LIN {X 0,Y 453.948,Z 433.148,A -85,B 0,C 180,E1 19620.953,E2 19620.953} C_VEL
LIN {X 0,Y 449.947,Z 427.727,A -85,B 0,C 180,E1 19618.536,E2 19618.536} C_VEL
LIN {X 0,Y 445.616,Z 421.973,A -85,B 0,C 180,E1 19615.625,E2 19615.625} C_VEL
LIN {X 0,Y 442.629,Z 417.979,A -85,B 0,C 180,E1 19613.319,E2 19613.319} C_VEL
LIN {X 0,Y 441.414,Z 416.212,A -85,B 0,C 180,E1 19612.32,E2 19612.32} C_VEL
LIN {X 0,Y 438.487,Z 412.431,A -85,B 0,C 180,E1 19609.754,E2 19609.754} C_VEL
LIN {X 0,Y 437.49,Z 410.574,A -85,B 0,C 180,E1 19608.658,E2 19608.658} C_VEL
LIN {X 0,Y 434.499,Z 406.882,A -85,B 0,C 180,E1 19605.473,E2 19605.473} C_VEL
LIN {X 0,Y 433.389,Z 405.057,A -85,B 0,C 180,E1 19604.065,E2 19604.065} C_VEL
LIN {X 0,Y 430.291,Z 402.854,A -85,B 0,C 180,E1 19600.026,E2 19600.026} C_VEL
LIN {X 0,Y 428.498,Z 399.899,A -85,B 0,C 180,E1 19596.497,E2 19596.497} C_VEL
LIN {X 0,Y 427.919,Z 398.821,A -85,B 0,C 180,E1 19594.98,E2 19594.98} C_VEL
LIN {X 0,Y 426.399,Z 397.892,A -85,B 0,C 180,E1 19590.961,E2 19590.961} C_VEL
LIN {X 0,Y 425.533,Z 397.406,A -85,B 0,C 180,E1 19586.482,E2 19586.482} C_VEL
LIN {X 0,Y 425.524,Z 397.366,A -85,B 0,C 180,E1 19581.704,E2 19581.704} C_VEL
LIN {X 0,Y 426.383,Z 397.854,A -85,B 0,C 180,E1 19577.222,E2 19577.222} C_VEL
LIN {X 0,Y 428.081,Z 398.875,A -85,B 0,C 180,E1 19573.002,E2 19573.002} C_VEL
LIN {X 0,Y 430.356,Z 402.874,A -85,B 0,C 180,E1 19568.465,E2 19568.465} C_VEL
LIN {X 0,Y 433.58,Z 405.087,A -85,B 0,C 180,E1 19564.562,E2 19564.562} C_VEL
LIN {X 0,Y 434.467,Z 405.993,A -85,B 0,C 180,E1 19563.639,E2 19563.639} C_VEL
LIN {X 0,Y 436.45,Z 409.448,A -85,B 0,C 180,E1 19561.412,E2 19561.412} C_VEL
LIN {X 0,Y 440.205,Z 412.266,A -85,B 0,C 180,E1 19558.341,E2 19558.341} C_VEL
LIN {X 0,Y 442.471,Z 415.992,A -85,B 0,C 180,E1 19556.507,E2 19556.507} C_VEL
LIN {X 0,Y 445.89,Z 418.808,A -85,B 0,C 180,E1 19554.263,E2 19554.263} C_VEL
LIN {X 0,Y 448.38,Z 422.573,A -85,B 0,C 180,E1 19552.597,E2 19552.597} C_VEL
LIN {X 0,Y 451.551,Z 425.296,A -85,B 0,C 180,E1 19550.859,E2 19550.859} C_VEL
LIN {X 0,Y 454.634,Z 429.505,A -85,B 0,C 180,E1 19549.129,E2 19549.129} C_VEL
LIN {X 0,Y 456.956,Z 431.699,A -85,B 0,C 180,E1 19548.003,E2 19548.003} C_VEL
LIN {X 0,Y 460.475,Z 436.08,A -85,B 0,C 180,E1 19546.306,E2 19546.306} C_VEL
LIN {X 0,Y 462.233,Z 437.873,A -85,B 0,C 180,E1 19545.527,E2 19545.527} C_VEL
LIN {X 0,Y 466.393,Z 442.761,A -85,B 0,C 180,E1 19543.767,E2 19543.767} C_VEL
LIN {X 0,Y 472.76,Z 450.553,A -85,B 0,C 180,E1 19541.251,E2 19541.251} C_VEL
LIN {X 0,Y 477.709,Z 456.627,A -85,B 0,C 180,E1 19539.457,E2 19539.457} C_VEL
LIN {X 0,Y 482.621,Z 462.669,A -85,B 0,C 180,E1 19537.805,E2 19537.805} C_VEL
LIN {X 0,Y 489.868,Z 471.652,A -85,B 0,C 180,E1 19535.534,E2 19535.534} C_VEL
LIN {X 0,Y 501.803,Z 487.082,A -85,B 0,C 180,E1 19532.17,E2 19532.17} C_VEL
LIN {X 0,Y 513.739,Z 503.433,A -85,B 0,C 180,E1 19529.164,E2 19529.164} C_VEL
LIN {X 0,Y 519.251,Z 511.432,A -85,B 0,C 180,E1 19527.864,E2 19527.864} C_VEL
LIN {X 0,Y 504.477,Z 710.205,A -85,B 0,C 180,E1 19524.562,E2 19524.562} C_VEL
LIN {X 0,Y 499.182,Z 782.061,A -85,B 0,C 180,E1 19523.337,E2 19523.337} C_VEL
LIN {X 0,Y 496,Z 810.118,A -85,B 0,C 180,E1 19522.672,E2 19522.672} C_VEL
LIN {X 0,Y 492.733,Z 832.872,A -85,B 0,C 180,E1 19521.983,E2 19521.983} C_VEL
LIN {X 0,Y 488.951,Z 855.104,A -85,B 0,C 180,E1 19521.169,E2 19521.169} C_VEL
LIN {X 0,Y 483.544,Z 882.162,A -85,B 0,C 180,E1 19519.967,E2 19519.967} C_VEL
LIN {X 0,Y 482.445,Z 886.921,A -85,B 0,C 180,E1 19519.725,E2 19519.725} C_VEL
LIN {X 0,Y 480.2,Z 894.101,A -85,B 0,C 180,E1 19519.451,E2 19519.451} C_VEL
LIN {X 0,Y 471.991,Z 912.002,A -85,B 0,C 180,E1 19519.007,E2 19519.007} C_VEL
LIN {X 0,Y 469.526,Z 918.813,A -85,B 0,C 180,E1 19518.673,E2 19518.673} C_VEL
LIN {X 0,Y 463.65,Z 939.58,A -85,B 0,C 180,E1 19517.251,E2 19517.251} C_VEL
LIN {X 0,Y 457.958,Z 958.139,A -85,B 0,C 180,E1 19515.794,E2 19515.794} C_VEL
LIN {X 0,Y 451.926,Z 976.561,A -85,B 0,C 180,E1 19514.149,E2 19514.149} C_VEL
LIN {X 0,Y 444.682,Z 997.402,A -85,B 0,C 180,E1 19512.016,E2 19512.016} C_VEL
LIN {X 0,Y 437.637,Z 1016.215,A -85,B 0,C 180,E1 19509.756,E2 19509.756} C_VEL
LIN {X 0,Y 431.782,Z 1031.379,A -85,B 0,C 180,E1 19507.68,E2 19507.68} C_VEL
LIN {X 0,Y 426.261,Z 1045.276,A -85,B 0,C 180,E1 19505.525,E2 19505.525} C_VEL
LIN {X 0,Y 420.181,Z 1060.321,A -85,B 0,C 180,E1 19502.873,E2 19502.873} C_VEL
LIN {X 0,Y 413.774,Z 1076.012,A -85,B 0,C 180,E1 19499.621,E2 19499.621} C_VEL
LIN {X 0,Y 409.258,Z 1087.2,A -85,B 0,C 180,E1 19496.931,E2 19496.931} C_VEL
LIN {X 0,Y 405.334,Z 1097.229,A -85,B 0,C 180,E1 19494.173,E2 19494.173} C_VEL
LIN {X 0,Y 401.802,Z 1106.699,A -85,B 0,C 180,E1 19491.161,E2 19491.161} C_VEL
LIN {X 0,Y 398.332,Z 1116.847,A -85,B 0,C 180,E1 19487.333,E2 19487.333} C_VEL
LIN {X 0,Y 396.087,Z 1124.106,A -85,B 0,C 180,E1 19483.965,E2 19483.965} C_VEL
LIN {X 0,Y 394.719,Z 1129.457,A -85,B 0,C 180,E1 19480.986,E2 19480.986} C_VEL
LIN {X 0,Y 393.77,Z 1133.759,A -85,B 0,C 180,E1 19478.079,E2 19478.079} C_VEL
LIN {X 0,Y 393.212,Z 1137.313,A -85,B 0,C 180,E1 19475.036,E2 19475.036} C_VEL
LIN {X 0,Y 392.895,Z 1140.115,A -85,B 0,C 180,E1 19471.789,E2 19471.789} C_VEL
LIN {X 0,Y 392.777,Z 1141.998,A -85,B 0,C 180,E1 19468.428,E2 19468.428} C_VEL
LIN {X 0,Y 392.756,Z 1142.857,A -85,B 0,C 180,E1 19464.518,E2 19464.518} C_VEL
LIN {X 0,Y 392.867,Z 1142.444,A -85,B 0,C 180,E1 19461.187,E2 19461.187} C_VEL
LIN {X 0,Y 393.077,Z 1141.179,A -85,B 0,C 180,E1 19458.08,E2 19458.08} C_VEL
LIN {X 0,Y 393.472,Z 1139.082,A -85,B 0,C 180,E1 19455.023,E2 19455.023} C_VEL
LIN {X 0,Y 394.158,Z 1136.173,A -85,B 0,C 180,E1 19452.006,E2 19452.006} C_VEL
LIN {X 0,Y 395.37,Z 1132.022,A -85,B 0,C 180,E1 19448.728,E2 19448.728} C_VEL
LIN {X 0,Y 397.737,Z 1125.255,A -85,B 0,C 180,E1 19444.614,E2 19444.614} C_VEL
LIN {X 0,Y 400.473,Z 1118.328,A -85,B 0,C 180,E1 19441.288,E2 19441.288} C_VEL
LIN {X 0,Y 403.679,Z 1110.94,A -85,B 0,C 180,E1 19438.297,E2 19438.297} C_VEL
LIN {X 0,Y 408.437,Z 1100.796,A -85,B 0,C 180,E1 19434.803,E2 19434.803} C_VEL
LIN {X 0,Y 414.124,Z 1088.742,A -85,B 0,C 180,E1 19431.391,E2 19431.391} C_VEL
LIN {X 0,Y 419.404,Z 1077.818,A -85,B 0,C 180,E1 19428.726,E2 19428.726} C_VEL
LIN {X 0,Y 426.356,Z 1063.666,A -85,B 0,C 180,E1 19425.744,E2 19425.744} C_VEL
LIN {X 0,Y 433.69,Z 1048.049,A -85,B 0,C 180,E1 19422.974,E2 19422.974} C_VEL
LIN {X 0,Y 440.644,Z 1033.015,A -85,B 0,C 180,E1 19420.652,E2 19420.652} C_VEL
LIN {X 0,Y 448.963,Z 1014.263,A -85,B 0,C 180,E1 19418.165,E2 19418.165} C_VEL
LIN {X 0,Y 456.181,Z 997.272,A -85,B 0,C 180,E1 19416.215,E2 19416.215} C_VEL
LIN {X 0,Y 464.592,Z 976.767,A -85,B 0,C 180,E1 19414.162,E2 19414.162} C_VEL
LIN {X 0,Y 473.151,Z 955.052,A -85,B 0,C 180,E1 19412.295,E2 19412.295} C_VEL
LIN {X 0,Y 483.358,Z 928.968,A -85,B 0,C 180,E1 19410.369,E2 19410.369} C_VEL
LIN {X 0,Y 492.594,Z 906.196,A -85,B 0,C 180,E1 19408.935,E2 19408.935} C_VEL
LIN {X 0,Y 480.962,Z 937.636,A -85,B 0,C 180,E1 19407.68,E2 19407.68} C_VEL
LIN {X 0,Y 469.639,Z 971.581,A -85,B 0,C 180,E1 19406.022,E2 19406.022} C_VEL
LIN {X 0,Y 459.445,Z 1005.778,A -85,B 0,C 180,E1 19404.054,E2 19404.054} C_VEL
LIN {X 0,Y 451.325,Z 1034.155,A -85,B 0,C 180,E1 19402.144,E2 19402.144} C_VEL
LIN {X 0,Y 444.279,Z 1059.225,A -85,B 0,C 180,E1 19400.225,E2 19400.225} C_VEL
LIN {X 0,Y 436.325,Z 1087.372,A -85,B 0,C 180,E1 19397.747,E2 19397.747} C_VEL
LIN {X 0,Y 430.123,Z 1109.071,A -85,B 0,C 180,E1 19395.533,E2 19395.533} C_VEL
LIN {X 0,Y 425.026,Z 1126.85,A -85,B 0,C 180,E1 19393.497,E2 19393.497} C_VEL
LIN {X 0,Y 420.318,Z 1143.268,A -85,B 0,C 180,E1 19391.401,E2 19391.401} C_VEL
LIN {X 0,Y 415.947,Z 1158.657,A -85,B 0,C 180,E1 19389.214,E2 19389.214} C_VEL
LIN {X 0,Y 411.781,Z 1173.547,A -85,B 0,C 180,E1 19386.853,E2 19386.853} C_VEL
LIN {X 0,Y 407.666,Z 1188.654,A -85,B 0,C 180,E1 19384.171,E2 19384.171} C_VEL
LIN {X 0,Y 403.227,Z 1205.646,A -85,B 0,C 180,E1 19380.718,E2 19380.718} C_VEL
LIN {X 0,Y 399.899,Z 1219.42,A -85,B 0,C 180,E1 19377.423,E2 19377.423} C_VEL
LIN {X 0,Y 397.604,Z 1230.079,A -85,B 0,C 180,E1 19374.515,E2 19374.515} C_VEL
LIN {X 0,Y 395.951,Z 1238.807,A -85,B 0,C 180,E1 19371.79,E2 19371.79} C_VEL
LIN {X 0,Y 394.633,Z 1246.816,A -85,B 0,C 180,E1 19368.924,E2 19368.924} C_VEL
LIN {X 0,Y 393.741,Z 1253.611,A -85,B 0,C 180,E1 19366.069,E2 19366.069} C_VEL
LIN {X 0,Y 393.177,Z 1259.28,A -85,B 0,C 180,E1 19363.231,E2 19363.231} C_VEL
LIN {X 0,Y 392.885,Z 1263.863,A -85,B 0,C 180,E1 19360.41,E2 19360.41} C_VEL
LIN {X 0,Y 392.748,Z 1267.365,A -85,B 0,C 180,E1 19357.607,E2 19357.607} C_VEL
LIN {X 0,Y 392.757,Z 1269.828,A -85,B 0,C 180,E1 19354.819,E2 19354.819} C_VEL
LIN {X 0,Y 392.748,Z 1271.271,A -85,B 0,C 180,E1 19352.043,E2 19352.043} C_VEL
LIN {X 0,Y 392.679,Z 1271.697,A -85,B 0,C 180,E1 19349.27,E2 19349.27} C_VEL
LIN {X 0,Y 392.664,Z 1271.06,A -85,B 0,C 180,E1 19346.35,E2 19346.35} C_VEL
LIN {X 0,Y 392.615,Z 1269.234,A -85,B 0,C 180,E1 19343.331,E2 19343.331} C_VEL
LIN {X 0,Y 392.612,Z 1266.454,A -85,B 0,C 180,E1 19340.472,E2 19340.472} C_VEL
LIN {X 0,Y 392.854,Z 1262.513,A -85,B 0,C 180,E1 19337.506,E2 19337.506} C_VEL
LIN {X 0,Y 393.394,Z 1257.173,A -85,B 0,C 180,E1 19334.37,E2 19334.37} C_VEL
LIN {X 0,Y 394.206,Z 1251.255,A -85,B 0,C 180,E1 19331.515,E2 19331.515} C_VEL
LIN {X 0,Y 395.584,Z 1243.879,A -85,B 0,C 180,E1 19328.5,E2 19328.5} C_VEL
LIN {X 0,Y 397.475,Z 1235.286,A -85,B 0,C 180,E1 19325.476,E2 19325.476} C_VEL
LIN {X 0,Y 400.437,Z 1223.887,A -85,B 0,C 180,E1 19322.003,E2 19322.003} C_VEL
LIN {X 0,Y 404.325,Z 1210.505,A -85,B 0,C 180,E1 19318.547,E2 19318.547} C_VEL
LIN {X 0,Y 408.307,Z 1197.936,A -85,B 0,C 180,E1 19315.72,E2 19315.72} C_VEL
LIN {X 0,Y 412.74,Z 1184.667,A -85,B 0,C 180,E1 19313.074,E2 19313.074} C_VEL
LIN {X 0,Y 418.106,Z 1169.084,A -85,B 0,C 180,E1 19310.319,E2 19310.319} C_VEL
LIN {X 0,Y 425.297,Z 1148.513,A -85,B 0,C 180,E1 19307.183,E2 19307.183} C_VEL
LIN {X 0,Y 431.319,Z 1131.262,A -85,B 0,C 180,E1 19304.911,E2 19304.911} C_VEL
LIN {X 0,Y 437.323,Z 1113.852,A -85,B 0,C 180,E1 19302.88,E2 19302.88} C_VEL
LIN {X 0,Y 444.975,Z 1091.294,A -85,B 0,C 180,E1 19300.58,E2 19300.58} C_VEL
LIN {X 0,Y 452.039,Z 1069.183,A -85,B 0,C 180,E1 19298.665,E2 19298.665} C_VEL
LIN {X 0,Y 458.025,Z 1049.435,A -85,B 0,C 180,E1 19297.174,E2 19297.174} C_VEL
LIN {X 0,Y 464.142,Z 1028.035,A -85,B 0,C 180,E1 19295.767,E2 19295.767} C_VEL
LIN {X 0,Y 471.265,Z 1001.001,A -85,B 0,C 180,E1 19294.27,E2 19294.27} C_VEL
LIN {X 0,Y 476.888,Z 977.149,A -85,B 0,C 180,E1 19293.178,E2 19293.178} C_VEL
LIN {X 0,Y 481.753,Z 954.324,A -85,B 0,C 180,E1 19292.308,E2 19292.308} C_VEL
LIN {X 0,Y 487.028,Z 925.599,A -85,B 0,C 180,E1 19291.431,E2 19291.431} C_VEL
LIN {X 0,Y 490.713,Z 900.074,A -85,B 0,C 180,E1 19290.827,E2 19290.827} C_VEL
LIN {X 0,Y 493.212,Z 875.395,A -85,B 0,C 180,E1 19290.338,E2 19290.338} C_VEL
LIN {X 0,Y 509.514,Z 656.144,A -85,B 0,C 180,E1 19286.627,E2 19286.627} C_VEL
LIN {X 0,Y 518.868,Z 538.73,A -85,B 0,C 180,E1 19284.628,E2 19284.628} C_VEL
LIN {X 0,Y 507.782,Z 520.812,A -85,B 0,C 180,E1 19281.819,E2 19281.819} C_VEL
LIN {X 0,Y 497.209,Z 504.575,A -85,B 0,C 180,E1 19278.861,E2 19278.861} C_VEL
LIN {X 0,Y 488.167,Z 490.995,A -85,B 0,C 180,E1 19276.052,E2 19276.052} C_VEL
LIN {X 0,Y 479.123,Z 477.956,A -85,B 0,C 180,E1 19272.947,E2 19272.947} C_VEL
LIN {X 0,Y 470.861,Z 466.4,A -85,B 0,C 180,E1 19269.781,E2 19269.781} C_VEL
LIN {X 0,Y 463.811,Z 456.641,A -85,B 0,C 180,E1 19266.747,E2 19266.747} C_VEL
LIN {X 0,Y 459.946,Z 451.491,A -85,B 0,C 180,E1 19264.926,E2 19264.926} C_VEL
LIN {X 0,Y 455.971,Z 445.983,A -85,B 0,C 180,E1 19262.891,E2 19262.891} C_VEL
LIN {X 0,Y 452.054,Z 440.675,A -85,B 0,C 180,E1 19260.697,E2 19260.697} C_VEL
LIN {X 0,Y 448.138,Z 435.338,A -85,B 0,C 180,E1 19258.314,E2 19258.314} C_VEL
LIN {X 0,Y 443.954,Z 429.716,A -85,B 0,C 180,E1 19255.479,E2 19255.479} C_VEL
LIN {X 0,Y 440.861,Z 425.59,A -85,B 0,C 180,E1 19253.096,E2 19253.096} C_VEL
LIN {X 0,Y 439.746,Z 423.943,A -85,B 0,C 180,E1 19252.159,E2 19252.159} C_VEL
LIN {X 0,Y 436.762,Z 420.025,A -85,B 0,C 180,E1 19249.514,E2 19249.514} C_VEL
LIN {X 0,Y 435.782,Z 418.267,A -85,B 0,C 180,E1 19248.443,E2 19248.443} C_VEL
LIN {X 0,Y 432.811,Z 414.468,A -85,B 0,C 180,E1 19245.21,E2 19245.21} C_VEL
LIN {X 0,Y 431.791,Z 412.866,A -85,B 0,C 180,E1 19243.944,E2 19243.944} C_VEL
LIN {X 0,Y 428.75,Z 410.685,A -85,B 0,C 180,E1 19239.951,E2 19239.951} C_VEL
LIN {X 0,Y 426.926,Z 407.628,A -85,B 0,C 180,E1 19236.31,E2 19236.31} C_VEL
LIN {X 0,Y 426.294,Z 406.597,A -85,B 0,C 180,E1 19234.73,E2 19234.73} C_VEL
LIN {X 0,Y 424.81,Z 405.705,A -85,B 0,C 180,E1 19230.687,E2 19230.687} C_VEL
LIN {X 0,Y 424.011,Z 405.252,A -85,B 0,C 180,E1 19226.184,E2 19226.184} C_VEL
LIN {X 0,Y 424.04,Z 405.22,A -85,B 0,C 180,E1 19221.5,E2 19221.5} C_VEL
LIN {X 0,Y 424.954,Z 405.761,A -85,B 0,C 180,E1 19217.033,E2 19217.033} C_VEL
LIN {X 0,Y 426.587,Z 406.753,A -85,B 0,C 180,E1 19213.004,E2 19213.004} C_VEL
LIN {X 0,Y 428.87,Z 410.741,A -85,B 0,C 180,E1 19208.498,E2 19208.498} C_VEL
LIN {X 0,Y 432.159,Z 412.977,A -85,B 0,C 180,E1 19204.531,E2 19204.531} C_VEL
LIN {X 0,Y 432.888,Z 413.863,A -85,B 0,C 180,E1 19203.743,E2 19203.743} C_VEL
LIN {X 0,Y 434.956,Z 417.333,A -85,B 0,C 180,E1 19201.455,E2 19201.455} C_VEL
LIN {X 0,Y 438.558,Z 420.075,A -85,B 0,C 180,E1 19198.498,E2 19198.498} C_VEL
LIN {X 0,Y 440.911,Z 423.804,A -85,B 0,C 180,E1 19196.615,E2 19196.615} C_VEL
LIN {X 0,Y 444.168,Z 426.588,A -85,B 0,C 180,E1 19194.434,E2 19194.434} C_VEL
LIN {X 0,Y 446.782,Z 430.378,A -85,B 0,C 180,E1 19192.709,E2 19192.709} C_VEL
LIN {X 0,Y 449.707,Z 432.919,A -85,B 0,C 180,E1 19191.078,E2 19191.078} C_VEL
LIN {X 0,Y 452.949,Z 437.251,A -85,B 0,C 180,E1 19189.27,E2 19189.27} C_VEL
LIN {X 0,Y 455.084,Z 439.332,A -85,B 0,C 180,E1 19188.216,E2 19188.216} C_VEL
LIN {X 0,Y 458.75,Z 443.799,A -85,B 0,C 180,E1 19186.458,E2 19186.458} C_VEL
LIN {X 0,Y 460.451,Z 445.673,A -85,B 0,C 180,E1 19185.685,E2 19185.685} C_VEL
LIN {X 0,Y 465.727,Z 451.979,A -85,B 0,C 180,E1 19183.45,E2 19183.45} C_VEL
LIN {X 0,Y 470.69,Z 458.055,A -85,B 0,C 180,E1 19181.487,E2 19181.487} C_VEL
LIN {X 0,Y 475.57,Z 464.047,A -85,B 0,C 180,E1 19179.714,E2 19179.714} C_VEL
LIN {X 0,Y 480.718,Z 470.467,A -85,B 0,C 180,E1 19177.957,E2 19177.957} C_VEL
LIN {X 0,Y 487.565,Z 479.019,A -85,B 0,C 180,E1 19175.796,E2 19175.796} C_VEL
LIN {X 0,Y 499.253,Z 494.246,A -85,B 0,C 180,E1 19172.462,E2 19172.462} C_VEL
LIN {X 0,Y 510.969,Z 510.428,A -85,B 0,C 180,E1 19169.471,E2 19169.471} C_VEL
LIN {X 0,Y 514.772,Z 516.195,A -85,B 0,C 180,E1 19168.55,E2 19168.55} C_VEL
LIN {X 0,Y 499.152,Z 719.913,A -85,B 0,C 180,E1 19165.148,E2 19165.148} C_VEL
LIN {X 0,Y 494.271,Z 783.622,A -85,B 0,C 180,E1 19164.051,E2 19164.051} C_VEL
LIN {X 0,Y 490.995,Z 811.533,A -85,B 0,C 180,E1 19163.381,E2 19163.381} C_VEL
LIN {X 0,Y 487.607,Z 834.455,A -85,B 0,C 180,E1 19162.681,E2 19162.681} C_VEL
LIN {X 0,Y 483.417,Z 858.306,A -85,B 0,C 180,E1 19161.795,E2 19161.795} C_VEL
LIN {X 0,Y 477.652,Z 885.781,A -85,B 0,C 180,E1 19160.542,E2 19160.542} C_VEL
LIN {X 0,Y 472.591,Z 906.898,A -85,B 0,C 180,E1 19159.393,E2 19159.393} C_VEL
LIN {X 0,Y 469.526,Z 918.813,A -85,B 0,C 180,E1 19158.673,E2 19158.673} C_VEL
LIN {X 0,Y 466.992,Z 925.701,A -85,B 0,C 180,E1 19158.318,E2 19158.318} C_VEL
LIN {X 0,Y 458.052,Z 942.989,A -85,B 0,C 180,E1 19157.685,E2 19157.685} C_VEL
LIN {X 0,Y 455.462,Z 949.44,A -85,B 0,C 180,E1 19157.291,E2 19157.291} C_VEL
LIN {X 0,Y 448.162,Z 971.708,A -85,B 0,C 180,E1 19155.398,E2 19155.398} C_VEL
LIN {X 0,Y 442.104,Z 988.918,A -85,B 0,C 180,E1 19153.713,E2 19153.713} C_VEL
LIN {X 0,Y 436.029,Z 1005.301,A -85,B 0,C 180,E1 19151.897,E2 19151.897} C_VEL
LIN {X 0,Y 429.758,Z 1021.526,A -85,B 0,C 180,E1 19149.859,E2 19149.859} C_VEL
LIN {X 0,Y 422.197,Z 1040.463,A -85,B 0,C 180,E1 19147.113,E2 19147.113} C_VEL
LIN {X 0,Y 415.633,Z 1056.182,A -85,B 0,C 180,E1 19144.441,E2 19144.441} C_VEL
LIN {X 0,Y 410.447,Z 1068.522,A -85,B 0,C 180,E1 19142.042,E2 19142.042} C_VEL
LIN {X 0,Y 405.407,Z 1080.465,A -85,B 0,C 180,E1 19139.404,E2 19139.404} C_VEL
LIN {X 0,Y 400.057,Z 1093.546,A -85,B 0,C 180,E1 19136.078,E2 19136.078} C_VEL
LIN {X 0,Y 395.444,Z 1105.037,A -85,B 0,C 180,E1 19132.557,E2 19132.557} C_VEL
LIN {X 0,Y 392.402,Z 1113.228,A -85,B 0,C 180,E1 19129.632,E2 19129.632} C_VEL
LIN {X 0,Y 389.901,Z 1120.518,A -85,B 0,C 180,E1 19126.586,E2 19126.586} C_VEL
LIN {X 0,Y 387.968,Z 1126.813,A -85,B 0,C 180,E1 19123.482,E2 19123.482} C_VEL
LIN {X 0,Y 386.417,Z 1133.084,A -85,B 0,C 180,E1 19119.728,E2 19119.728} C_VEL
LIN {X 0,Y 385.422,Z 1138.027,A -85,B 0,C 180,E1 19115.709,E2 19115.709} C_VEL
LIN {X 0,Y 385.041,Z 1140.904,A -85,B 0,C 180,E1 19112.517,E2 19112.517} C_VEL
LIN {X 0,Y 384.895,Z 1142.77,A -85,B 0,C 180,E1 19109.512,E2 19109.512} C_VEL
LIN {X 0,Y 384.832,Z 1143.831,A -85,B 0,C 180,E1 19106.545,E2 19106.545} C_VEL
LIN {X 0,Y 384.884,Z 1144.122,A -85,B 0,C 180,E1 19103.746,E2 19103.746} C_VEL
LIN {X 0,Y 384.993,Z 1143.683,A -85,B 0,C 180,E1 19100.778,E2 19100.778} C_VEL
LIN {X 0,Y 385.233,Z 1142.497,A -85,B 0,C 180,E1 19097.835,E2 19097.835} C_VEL
LIN {X 0,Y 385.675,Z 1140.418,A -85,B 0,C 180,E1 19094.719,E2 19094.719} C_VEL
LIN {X 0,Y 386.514,Z 1137.205,A -85,B 0,C 180,E1 19091.352,E2 19091.352} C_VEL
LIN {X 0,Y 388.2,Z 1132.139,A -85,B 0,C 180,E1 19087.399,E2 19087.399} C_VEL
LIN {X 0,Y 390.641,Z 1125.75,A -85,B 0,C 180,E1 19083.669,E2 19083.669} C_VEL
LIN {X 0,Y 393.382,Z 1119.366,A -85,B 0,C 180,E1 19080.583,E2 19080.583} C_VEL
LIN {X 0,Y 397.201,Z 1111.219,A -85,B 0,C 180,E1 19077.259,E2 19077.259} C_VEL
LIN {X 0,Y 402.764,Z 1099.869,A -85,B 0,C 180,E1 19073.443,E2 19073.443} C_VEL
LIN {X 0,Y 407.935,Z 1089.631,A -85,B 0,C 180,E1 19070.548,E2 19070.548} C_VEL
LIN {X 0,Y 413.544,Z 1078.673,A -85,B 0,C 180,E1 19067.857,E2 19067.857} C_VEL
LIN {X 0,Y 421.484,Z 1063.066,A -85,B 0,C 180,E1 19064.591,E2 19064.591} C_VEL
LIN {X 0,Y 428.184,Z 1049.59,A -85,B 0,C 180,E1 19062.187,E2 19062.187} C_VEL
LIN {X 0,Y 435.869,Z 1033.871,A -85,B 0,C 180,E1 19059.733,E2 19059.733} C_VEL
LIN {X 0,Y 444.57,Z 1015.144,A -85,B 0,C 180,E1 19057.241,E2 19057.241} C_VEL
LIN {X 0,Y 452.884,Z 996.858,A -85,B 0,C 180,E1 19055.128,E2 19055.128} C_VEL
LIN {X 0,Y 463.019,Z 973.63,A -85,B 0,C 180,E1 19052.835,E2 19052.835} C_VEL
LIN {X 0,Y 474.672,Z 946.973,A -85,B 0,C 180,E1 19050.606,E2 19050.606} C_VEL
LIN {X 0,Y 484.052,Z 926.526,A -85,B 0,C 180,E1 19049.128,E2 19049.128} C_VEL
LIN {X 0,Y 473.909,Z 950.996,A -85,B 0,C 180,E1 19048.012,E2 19048.012} C_VEL
LIN {X 0,Y 462.82,Z 980.985,A -85,B 0,C 180,E1 19046.402,E2 19046.402} C_VEL
LIN {X 0,Y 451.011,Z 1017.128,A -85,B 0,C 180,E1 19044.125,E2 19044.125} C_VEL
LIN {X 0,Y 441.189,Z 1049.264,A -85,B 0,C 180,E1 19041.747,E2 19041.747} C_VEL
LIN {X 0,Y 433.977,Z 1073.393,A -85,B 0,C 180,E1 19039.695,E2 19039.695} C_VEL
LIN {X 0,Y 426.427,Z 1099.016,A -85,B 0,C 180,E1 19037.215,E2 19037.215} C_VEL
LIN {X 0,Y 419.399,Z 1122.234,A -85,B 0,C 180,E1 19034.596,E2 19034.596} C_VEL
LIN {X 0,Y 414.118,Z 1139.858,A -85,B 0,C 180,E1 19032.348,E2 19032.348} C_VEL
LIN {X 0,Y 409.356,Z 1155.854,A -85,B 0,C 180,E1 19030.068,E2 19030.068} C_VEL
LIN {X 0,Y 405.077,Z 1170.456,A -85,B 0,C 180,E1 19027.745,E2 19027.745} C_VEL
LIN {X 0,Y 401.162,Z 1184.09,A -85,B 0,C 180,E1 19025.327,E2 19025.327} C_VEL
LIN {X 0,Y 397.4,Z 1197.937,A -85,B 0,C 180,E1 19022.577,E2 19022.577} C_VEL
LIN {X 0,Y 393.526,Z 1212.84,A -85,B 0,C 180,E1 19019.198,E2 19019.198} C_VEL
LIN {X 0,Y 390.283,Z 1226.724,A -85,B 0,C 180,E1 19015.493,E2 19015.493} C_VEL
LIN {X 0,Y 388.265,Z 1236.659,A -85,B 0,C 180,E1 19012.402,E2 19012.402} C_VEL
LIN {X 0,Y 386.822,Z 1245.076,A -85,B 0,C 180,E1 19009.354,E2 19009.354} C_VEL
LIN {X 0,Y 385.867,Z 1252.051,A -85,B 0,C 180,E1 19006.406,E2 19006.406} C_VEL
LIN {X 0,Y 385.276,Z 1257.781,A -85,B 0,C 180,E1 19003.507,E2 19003.507} C_VEL
LIN {X 0,Y 384.989,Z 1262.193,A -85,B 0,C 180,E1 19000.777,E2 19000.777} C_VEL
LIN {X 0,Y 384.84,Z 1265.964,A -85,B 0,C 180,E1 18997.765,E2 18997.765} C_VEL
LIN {X 0,Y 384.858,Z 1268.485,A -85,B 0,C 180,E1 18994.918,E2 18994.918} C_VEL
LIN {X 0,Y 384.852,Z 1270.006,A -85,B 0,C 180,E1 18991.935,E2 18991.935} C_VEL
LIN {X 0,Y 384.785,Z 1270.396,A -85,B 0,C 180,E1 18989.107,E2 18989.107} C_VEL
LIN {X 0,Y 384.76,Z 1269.786,A -85,B 0,C 180,E1 18986.275,E2 18986.275} C_VEL
LIN {X 0,Y 384.697,Z 1268.043,A -85,B 0,C 180,E1 18983.283,E2 18983.283} C_VEL
LIN {X 0,Y 384.693,Z 1265.192,A -85,B 0,C 180,E1 18980.273,E2 18980.273} C_VEL
LIN {X 0,Y 384.929,Z 1261.231,A -85,B 0,C 180,E1 18977.244,E2 18977.244} C_VEL
LIN {X 0,Y 385.467,Z 1256.147,A -85,B 0,C 180,E1 18974.195,E2 18974.195} C_VEL
LIN {X 0,Y 386.373,Z 1249.913,A -85,B 0,C 180,E1 18971.126,E2 18971.126} C_VEL
LIN {X 0,Y 387.821,Z 1242.517,A -85,B 0,C 180,E1 18968.048,E2 18968.048} C_VEL
LIN {X 0,Y 389.932,Z 1233.445,A -85,B 0,C 180,E1 18964.807,E2 18964.807} C_VEL
LIN {X 0,Y 393.449,Z 1220.752,A -85,B 0,C 180,E1 18960.954,E2 18960.954} C_VEL
LIN {X 0,Y 397.45,Z 1207.679,A -85,B 0,C 180,E1 18957.598,E2 18957.598} C_VEL
LIN {X 0,Y 401.703,Z 1194.933,A -85,B 0,C 180,E1 18954.727,E2 18954.727} C_VEL
LIN {X 0,Y 406.957,Z 1179.922,A -85,B 0,C 180,E1 18951.746,E2 18951.746} C_VEL
LIN {X 0,Y 413.766,Z 1160.94,A -85,B 0,C 180,E1 18948.516,E2 18948.516} C_VEL
LIN {X 0,Y 419.667,Z 1144.656,A -85,B 0,C 180,E1 18946.106,E2 18946.106} C_VEL
LIN {X 0,Y 425.669,Z 1128.075,A -85,B 0,C 180,E1 18943.933,E2 18943.933} C_VEL
LIN {X 0,Y 433.016,Z 1107.569,A -85,B 0,C 180,E1 18941.57,E2 18941.57} C_VEL
LIN {X 0,Y 440.561,Z 1085.37,A -85,B 0,C 180,E1 18939.396,E2 18939.396} C_VEL
LIN {X 0,Y 446.678,Z 1066.656,A -85,B 0,C 180,E1 18937.798,E2 18937.798} C_VEL
LIN {X 0,Y 452.867,Z 1046.76,A -85,B 0,C 180,E1 18936.305,E2 18936.305} C_VEL
LIN {X 0,Y 460.208,Z 1021.636,A -85,B 0,C 180,E1 18934.679,E2 18934.679} C_VEL
LIN {X 0,Y 466.794,Z 996.596,A -85,B 0,C 180,E1 18933.344,E2 18933.344} C_VEL
LIN {X 0,Y 472.008,Z 974.922,A -85,B 0,C 180,E1 18932.367,E2 18932.367} C_VEL
LIN {X 0,Y 477.145,Z 951.23,A -85,B 0,C 180,E1 18931.473,E2 18931.473} C_VEL
LIN {X 0,Y 482.513,Z 922.024,A -85,B 0,C 180,E1 18930.606,E2 18930.606} C_VEL
LIN {X 0,Y 485.959,Z 898.369,A -85,B 0,C 180,E1 18930.051,E2 18930.051} C_VEL
LIN {X 0,Y 488.459,Z 874.081,A -85,B 0,C 180,E1 18929.57,E2 18929.57} C_VEL
LIN {X 0,Y 505.172,Z 656.069,A -85,B 0,C 180,E1 18925.864,E2 18925.864} C_VEL
LIN {X 0,Y 514.489,Z 543.125,A -85,B 0,C 180,E1 18923.935,E2 18923.935} C_VEL
LIN {X 0,Y 504.01,Z 526.227,A -85,B 0,C 180,E1 18921.227,E2 18921.227} C_VEL
LIN {X 0,Y 494.313,Z 511.183,A -85,B 0,C 180,E1 18918.455,E2 18918.455} C_VEL
LIN {X 0,Y 485.424,Z 497.743,A -85,B 0,C 180,E1 18915.655,E2 18915.655} C_VEL
LIN {X 0,Y 476.505,Z 484.809,A -85,B 0,C 180,E1 18912.544,E2 18912.544} C_VEL
LIN {X 0,Y 468.459,Z 473.405,A -85,B 0,C 180,E1 18909.398,E2 18909.398} C_VEL
LIN {X 0,Y 461.241,Z 463.344,A -85,B 0,C 180,E1 18906.223,E2 18906.223} C_VEL
LIN {X 0,Y 457.771,Z 458.725,A -85,B 0,C 180,E1 18904.573,E2 18904.573} C_VEL
LIN {X 0,Y 454.075,Z 453.52,A -85,B 0,C 180,E1 18902.65,E2 18902.65} C_VEL
LIN {X 0,Y 450.157,Z 448.208,A -85,B 0,C 180,E1 18900.445,E2 18900.445} C_VEL
LIN {X 0,Y 446.212,Z 442.819,A -85,B 0,C 180,E1 18898.017,E2 18898.017} C_VEL
LIN {X 0,Y 442.295,Z 437.46,A -85,B 0,C 180,E1 18895.332,E2 18895.332} C_VEL
LIN {X 0,Y 439.177,Z 433.344,A -85,B 0,C 180,E1 18892.938,E2 18892.938} C_VEL
LIN {X 0,Y 438.08,Z 431.674,A -85,B 0,C 180,E1 18891.997,E2 18891.997} C_VEL
LIN {X 0,Y 435.045,Z 427.619,A -85,B 0,C 180,E1 18889.271,E2 18889.271} C_VEL
LIN {X 0,Y 434.013,Z 425.898,A -85,B 0,C 180,E1 18888.168,E2 18888.168} C_VEL
LIN {X 0,Y 431.171,Z 422.159,A -85,B 0,C 180,E1 18885.015,E2 18885.015} C_VEL
LIN {X 0,Y 430.13,Z 420.639,A -85,B 0,C 180,E1 18883.751,E2 18883.751} C_VEL
LIN {X 0,Y 427.124,Z 418.403,A -85,B 0,C 180,E1 18879.729,E2 18879.729} C_VEL
LIN {X 0,Y 425.323,Z 415.232,A -85,B 0,C 180,E1 18876.002,E2 18876.002} C_VEL
LIN {X 0,Y 424.294,Z 414.017,A -85,B 0,C 180,E1 18873.551,E2 18873.551} C_VEL
LIN {X 0,Y 422.9,Z 413.377,A -85,B 0,C 180,E1 18868.973,E2 18868.973} C_VEL
LIN {X 0,Y 422.39,Z 413.023,A -85,B 0,C 180,E1 18864.385,E2 18864.385} C_VEL
LIN {X 0,Y 422.734,Z 413.245,A -85,B 0,C 180,E1 18860.027,E2 18860.027} C_VEL
LIN {X 0,Y 424.141,Z 413.928,A -85,B 0,C 180,E1 18855.18,E2 18855.18} C_VEL
LIN {X 0,Y 425.287,Z 414.934,A -85,B 0,C 180,E1 18852.617,E2 18852.617} C_VEL
LIN {X 0,Y 427.301,Z 418.508,A -85,B 0,C 180,E1 18848.666,E2 18848.666} C_VEL
LIN {X 0,Y 430.566,Z 420.78,A -85,B 0,C 180,E1 18844.677,E2 18844.677} C_VEL
LIN {X 0,Y 431.271,Z 421.631,A -85,B 0,C 180,E1 18843.899,E2 18843.899} C_VEL
LIN {X 0,Y 433.373,Z 425.115,A -85,B 0,C 180,E1 18841.583,E2 18841.583} C_VEL
LIN {X 0,Y 436.924,Z 427.897,A -85,B 0,C 180,E1 18838.648,E2 18838.648} C_VEL
LIN {X 0,Y 439.502,Z 431.785,A -85,B 0,C 180,E1 18836.607,E2 18836.607} C_VEL
LIN {X 0,Y 442.399,Z 434.253,A -85,B 0,C 180,E1 18834.645,E2 18834.645} C_VEL
LIN {X 0,Y 445.232,Z 438.231,A -85,B 0,C 180,E1 18832.792,E2 18832.792} C_VEL
LIN {X 0,Y 447.981,Z 440.73,A -85,B 0,C 180,E1 18831.231,E2 18831.231} C_VEL
LIN {X 0,Y 451.419,Z 445.139,A -85,B 0,C 180,E1 18829.336,E2 18829.336} C_VEL
LIN {X 0,Y 453.213,Z 446.945,A -85,B 0,C 180,E1 18828.435,E2 18828.435} C_VEL
LIN {X 0,Y 457.028,Z 451.517,A -85,B 0,C 180,E1 18826.611,E2 18826.611} C_VEL
LIN {X 0,Y 458.75,Z 453.569,A -85,B 0,C 180,E1 18825.81,E2 18825.81} C_VEL
LIN {X 0,Y 463.721,Z 459.508,A -85,B 0,C 180,E1 18823.685,E2 18823.685} C_VEL
LIN {X 0,Y 468.559,Z 465.462,A -85,B 0,C 180,E1 18821.753,E2 18821.753} C_VEL
LIN {X 0,Y 473.683,Z 471.814,A -85,B 0,C 180,E1 18819.875,E2 18819.875} C_VEL
LIN {X 0,Y 481.091,Z 480.954,A -85,B 0,C 180,E1 18817.374,E2 18817.374} C_VEL
LIN {X 0,Y 493.084,Z 496.573,A -85,B 0,C 180,E1 18813.753,E2 18813.753} C_VEL
LIN {X 0,Y 505.119,Z 513.052,A -85,B 0,C 180,E1 18810.539,E2 18810.539} C_VEL
LIN {X 0,Y 510.335,Z 520.769,A -85,B 0,C 180,E1 18809.248,E2 18809.248} C_VEL
LIN {X 0,Y 493.695,Z 731.672,A -85,B 0,C 180,E1 18805.712,E2 18805.712} C_VEL
LIN {X 0,Y 489.4,Z 785.641,A -85,B 0,C 180,E1 18804.771,E2 18804.771} C_VEL
LIN {X 0,Y 486.068,Z 812.89,A -85,B 0,C 180,E1 18804.107,E2 18804.107} C_VEL
LIN {X 0,Y 482.643,Z 835.454,A -85,B 0,C 180,E1 18803.413,E2 18803.413} C_VEL
LIN {X 0,Y 478.352,Z 859.289,A -85,B 0,C 180,E1 18802.524,E2 18802.524} C_VEL
LIN {X 0,Y 472.433,Z 886.808,A -85,B 0,C 180,E1 18801.263,E2 18801.263} C_VEL
LIN {X 0,Y 467.413,Z 907.287,A -85,B 0,C 180,E1 18800.146,E2 18800.146} C_VEL
LIN {X 0,Y 462.317,Z 926.17,A -85,B 0,C 180,E1 18798.965,E2 18798.965} C_VEL
LIN {X 0,Y 456.443,Z 946.091,A -85,B 0,C 180,E1 18797.546,E2 18797.546} C_VEL
LIN {X 0,Y 455.462,Z 949.44,A -85,B 0,C 180,E1 18797.291,E2 18797.291} C_VEL
LIN {X 0,Y 452.811,Z 955.95,A -85,B 0,C 180,E1 18796.875,E2 18796.875} C_VEL
LIN {X 0,Y 442.718,Z 973.283,A -85,B 0,C 180,E1 18795.978,E2 18795.978} C_VEL
LIN {X 0,Y 440.339,Z 978.566,A -85,B 0,C 180,E1 18795.558,E2 18795.558} C_VEL
LIN {X 0,Y 432.529,Z 999.936,A -85,B 0,C 180,E1 18793.343,E2 18793.343} C_VEL
LIN {X 0,Y 425.436,Z 1017.932,A -85,B 0,C 180,E1 18791.153,E2 18791.153} C_VEL
LIN {X 0,Y 419.196,Z 1033.168,A -85,B 0,C 180,E1 18789.036,E2 18789.036} C_VEL
LIN {X 0,Y 413.3,Z 1047.189,A -85,B 0,C 180,E1 18786.829,E2 18786.829} C_VEL
LIN {X 0,Y 407.237,Z 1061.332,A -85,B 0,C 180,E1 18784.303,E2 18784.303} C_VEL
LIN {X 0,Y 400.026,Z 1077.938,A -85,B 0,C 180,E1 18780.83,E2 18780.83} C_VEL
LIN {X 0,Y 395.042,Z 1089.475,A -85,B 0,C 180,E1 18777.987,E2 18777.987} C_VEL
LIN {X 0,Y 390.872,Z 1099.334,A -85,B 0,C 180,E1 18775.201,E2 18775.201} C_VEL
LIN {X 0,Y 387.367,Z 1107.943,A -85,B 0,C 180,E1 18772.415,E2 18772.415} C_VEL
LIN {X 0,Y 384.313,Z 1115.951,A -85,B 0,C 180,E1 18769.426,E2 18769.426} C_VEL
LIN {X 0,Y 381.343,Z 1124.714,A -85,B 0,C 180,E1 18765.568,E2 18765.568} C_VEL
LIN {X 0,Y 379.268,Z 1131.534,A -85,B 0,C 180,E1 18761.748,E2 18761.748} C_VEL
LIN {X 0,Y 378.15,Z 1136.073,A -85,B 0,C 180,E1 18758.611,E2 18758.611} C_VEL
LIN {X 0,Y 377.496,Z 1139.683,A -85,B 0,C 180,E1 18755.456,E2 18755.456} C_VEL
LIN {X 0,Y 377.147,Z 1142.337,A -85,B 0,C 180,E1 18752.381,E2 18752.381} C_VEL
LIN {X 0,Y 376.994,Z 1144.13,A -85,B 0,C 180,E1 18749.385,E2 18749.385} C_VEL
LIN {X 0,Y 376.943,Z 1145.146,A -85,B 0,C 180,E1 18746.465,E2 18746.465} C_VEL
LIN {X 0,Y 376.995,Z 1145.443,A -85,B 0,C 180,E1 18743.609,E2 18743.609} C_VEL
LIN {X 0,Y 377.123,Z 1145.027,A -85,B 0,C 180,E1 18740.624,E2 18740.624} C_VEL
LIN {X 0,Y 377.406,Z 1143.786,A -85,B 0,C 180,E1 18737.492,E2 18737.492} C_VEL
LIN {X 0,Y 377.89,Z 1141.759,A -85,B 0,C 180,E1 18734.402,E2 18734.402} C_VEL
LIN {X 0,Y 378.83,Z 1138.536,A -85,B 0,C 180,E1 18730.934,E2 18730.934} C_VEL
LIN {X 0,Y 380.826,Z 1133.008,A -85,B 0,C 180,E1 18726.634,E2 18726.634} C_VEL
LIN {X 0,Y 383.274,Z 1127.13,A -85,B 0,C 180,E1 18723.141,E2 18723.141} C_VEL
LIN {X 0,Y 386.369,Z 1120.446,A -85,B 0,C 180,E1 18719.852,E2 18719.852} C_VEL
LIN {X 0,Y 391.072,Z 1111.136,A -85,B 0,C 180,E1 18716.042,E2 18716.042} C_VEL
LIN {X 0,Y 396.374,Z 1100.835,A -85,B 0,C 180,E1 18712.608,E2 18712.608} C_VEL
LIN {X 0,Y 401.594,Z 1091.108,A -85,B 0,C 180,E1 18709.818,E2 18709.818} C_VEL
LIN {X 0,Y 408.794,Z 1077.93,A -85,B 0,C 180,E1 18706.564,E2 18706.564} C_VEL
LIN {X 0,Y 416.141,Z 1063.96,A -85,B 0,C 180,E1 18703.673,E2 18703.673} C_VEL
LIN {X 0,Y 422.805,Z 1051.256,A -85,B 0,C 180,E1 18701.382,E2 18701.382} C_VEL
LIN {X 0,Y 431.282,Z 1034.917,A -85,B 0,C 180,E1 18698.797,E2 18698.797} C_VEL
LIN {X 0,Y 440.406,Z 1016.305,A -85,B 0,C 180,E1 18696.306,E2 18696.306} C_VEL
LIN {X 0,Y 450.409,Z 995.719,A -85,B 0,C 180,E1 18693.925,E2 18693.925} C_VEL
LIN {X 0,Y 462.521,Z 970.559,A -85,B 0,C 180,E1 18691.46,E2 18691.46} C_VEL
LIN {X 0,Y 474.819,Z 945.961,A -85,B 0,C 180,E1 18689.432,E2 18689.432} C_VEL
LIN {X 0,Y 475.495,Z 944.669,A -85,B 0,C 180,E1 18689.322,E2 18689.322} C_VEL
LIN {X 0,Y 464.741,Z 968.441,A -85,B 0,C 180,E1 18688.076,E2 18688.076} C_VEL
LIN {X 0,Y 453.781,Z 996.131,A -85,B 0,C 180,E1 18686.397,E2 18686.397} C_VEL
LIN {X 0,Y 441.777,Z 1030.265,A -85,B 0,C 180,E1 18684.011,E2 18684.011} C_VEL
LIN {X 0,Y 430.969,Z 1063.68,A -85,B 0,C 180,E1 18681.285,E2 18681.285} C_VEL
LIN {X 0,Y 423.71,Z 1086.509,A -85,B 0,C 180,E1 18679.141,E2 18679.141} C_VEL
LIN {X 0,Y 417.532,Z 1106.116,A -85,B 0,C 180,E1 18677.069,E2 18677.069} C_VEL
LIN {X 0,Y 411.277,Z 1126.076,A -85,B 0,C 180,E1 18674.698,E2 18674.698} C_VEL
LIN {X 0,Y 404.082,Z 1149.224,A -85,B 0,C 180,E1 18671.54,E2 18671.54} C_VEL
LIN {X 0,Y 398.767,Z 1166.498,A -85,B 0,C 180,E1 18668.818,E2 18668.818} C_VEL
LIN {X 0,Y 394.349,Z 1181.191,A -85,B 0,C 180,E1 18666.212,E2 18666.212} C_VEL
LIN {X 0,Y 390.511,Z 1194.424,A -85,B 0,C 180,E1 18663.577,E2 18663.577} C_VEL
LIN {X 0,Y 387.089,Z 1207.016,A -85,B 0,C 180,E1 18660.76,E2 18660.76} C_VEL
LIN {X 0,Y 383.941,Z 1219.365,A -85,B 0,C 180,E1 18657.617,E2 18657.617} C_VEL
LIN {X 0,Y 381.201,Z 1231.678,A -85,B 0,C 180,E1 18653.989,E2 18653.989} C_VEL
LIN {X 0,Y 379.135,Z 1242.546,A -85,B 0,C 180,E1 18650.136,E2 18650.136} C_VEL
LIN {X 0,Y 378.052,Z 1250.146,A -85,B 0,C 180,E1 18646.913,E2 18646.913} C_VEL
LIN {X 0,Y 377.386,Z 1256,A -85,B 0,C 180,E1 18643.952,E2 18643.952} C_VEL
LIN {X 0,Y 377.078,Z 1260.758,A -85,B 0,C 180,E1 18641.006,E2 18641.006} C_VEL
LIN {X 0,Y 376.936,Z 1264.563,A -85,B 0,C 180,E1 18637.928,E2 18637.928} C_VEL
LIN {X 0,Y 376.961,Z 1267.118,A -85,B 0,C 180,E1 18635.022,E2 18635.022} C_VEL
LIN {X 0,Y 376.963,Z 1268.631,A -85,B 0,C 180,E1 18632.128,E2 18632.128} C_VEL
LIN {X 0,Y 376.89,Z 1269.105,A -85,B 0,C 180,E1 18629.24,E2 18629.24} C_VEL
LIN {X 0,Y 376.858,Z 1268.497,A -85,B 0,C 180,E1 18626.197,E2 18626.197} C_VEL
LIN {X 0,Y 376.782,Z 1266.756,A -85,B 0,C 180,E1 18623.141,E2 18623.141} C_VEL
LIN {X 0,Y 376.782,Z 1263.895,A -85,B 0,C 180,E1 18620.067,E2 18620.067} C_VEL
LIN {X 0,Y 377.012,Z 1259.922,A -85,B 0,C 180,E1 18616.972,E2 18616.972} C_VEL
LIN {X 0,Y 377.571,Z 1254.823,A -85,B 0,C 180,E1 18613.856,E2 18613.856} C_VEL
LIN {X 0,Y 378.547,Z 1248.578,A -85,B 0,C 180,E1 18610.721,E2 18610.721} C_VEL
LIN {X 0,Y 380.152,Z 1240.754,A -85,B 0,C 180,E1 18607.418,E2 18607.418} C_VEL
LIN {X 0,Y 382.966,Z 1229.724,A -85,B 0,C 180,E1 18603.483,E2 18603.483} C_VEL
LIN {X 0,Y 386.512,Z 1217.541,A -85,B 0,C 180,E1 18599.877,E2 18599.877} C_VEL
LIN {X 0,Y 390.26,Z 1206.074,A -85,B 0,C 180,E1 18596.91,E2 18596.91} C_VEL
LIN {X 0,Y 394.423,Z 1194.031,A -85,B 0,C 180,E1 18594.155,E2 18594.155} C_VEL
LIN {X 0,Y 399.881,Z 1178.975,A -85,B 0,C 180,E1 18591.126,E2 18591.126} C_VEL
LIN {X 0,Y 407.082,Z 1159.661,A -85,B 0,C 180,E1 18587.796,E2 18587.796} C_VEL
LIN {X 0,Y 413.227,Z 1143.297,A -85,B 0,C 180,E1 18585.349,E2 18585.349} C_VEL
LIN {X 0,Y 419.432,Z 1126.712,A -85,B 0,C 180,E1 18583.158,E2 18583.158} C_VEL
LIN {X 0,Y 427.285,Z 1105.337,A -85,B 0,C 180,E1 18580.696,E2 18580.696} C_VEL
LIN {X 0,Y 435.007,Z 1083.157,A -85,B 0,C 180,E1 18578.529,E2 18578.529} C_VEL
LIN {X 0,Y 441.538,Z 1063.729,A -85,B 0,C 180,E1 18576.878,E2 18576.878} C_VEL
LIN {X 0,Y 448.463,Z 1042.048,A -85,B 0,C 180,E1 18575.273,E2 18575.273} C_VEL
LIN {X 0,Y 455.92,Z 1016.607,A -85,B 0,C 180,E1 18573.678,E2 18573.678} C_VEL
LIN {X 0,Y 461.846,Z 994.502,A -85,B 0,C 180,E1 18572.515,E2 18572.515} C_VEL
LIN {X 0,Y 467.217,Z 972.585,A -85,B 0,C 180,E1 18571.539,E2 18571.539} C_VEL
LIN {X 0,Y 473.093,Z 945.753,A -85,B 0,C 180,E1 18570.551,E2 18570.551} C_VEL
LIN {X 0,Y 477.995,Z 918.728,A -85,B 0,C 180,E1 18569.782,E2 18569.782} C_VEL
LIN {X 0,Y 481.429,Z 894.977,A -85,B 0,C 180,E1 18569.232,E2 18569.232} C_VEL
LIN {X 0,Y 484.416,Z 864.358,A -85,B 0,C 180,E1 18568.644,E2 18568.644} C_VEL
LIN {X 0,Y 500.034,Z 666.851,A -85,B 0,C 180,E1 18565.272,E2 18565.272} C_VEL
LIN {X 0,Y 510.163,Z 547.588,A -85,B 0,C 180,E1 18563.231,E2 18563.231} C_VEL
LIN {X 0,Y 499.915,Z 531.06,A -85,B 0,C 180,E1 18560.519,E2 18560.519} C_VEL
LIN {X 0,Y 489.766,Z 515.1,A -85,B 0,C 180,E1 18557.526,E2 18557.526} C_VEL
LIN {X 0,Y 480.618,Z 501.49,A -85,B 0,C 180,E1 18554.549,E2 18554.549} C_VEL
LIN {X 0,Y 471.591,Z 488.177,A -85,B 0,C 180,E1 18551.248,E2 18551.248} C_VEL
LIN {X 0,Y 463.794,Z 477.266,A -85,B 0,C 180,E1 18548.056,E2 18548.056} C_VEL
LIN {X 0,Y 457.117,Z 467.756,A -85,B 0,C 180,E1 18544.957,E2 18544.957} C_VEL
LIN {X 0,Y 451.789,Z 460.617,A -85,B 0,C 180,E1 18542.22,E2 18542.22} C_VEL
LIN {X 0,Y 448.146,Z 455.609,A -85,B 0,C 180,E1 18540.128,E2 18540.128} C_VEL
LIN {X 0,Y 444.438,Z 450.454,A -85,B 0,C 180,E1 18537.808,E2 18537.808} C_VEL
LIN {X 0,Y 440.46,Z 445.024,A -85,B 0,C 180,E1 18535.051,E2 18535.051} C_VEL
LIN {X 0,Y 437.272,Z 440.668,A -85,B 0,C 180,E1 18532.577,E2 18532.577} C_VEL
LIN {X 0,Y 435.775,Z 438.738,A -85,B 0,C 180,E1 18531.29,E2 18531.29} C_VEL
LIN {X 0,Y 432.982,Z 434.418,A -85,B 0,C 180,E1 18528.612,E2 18528.612} C_VEL
LIN {X 0,Y 429.493,Z 429.838,A -85,B 0,C 180,E1 18524.817,E2 18524.817} C_VEL
LIN {X 0,Y 428.636,Z 428.503,A -85,B 0,C 180,E1 18523.744,E2 18523.744} C_VEL
LIN {X 0,Y 425.505,Z 426.122,A -85,B 0,C 180,E1 18519.504,E2 18519.504} C_VEL
LIN {X 0,Y 423.733,Z 422.9,A -85,B 0,C 180,E1 18515.758,E2 18515.758} C_VEL
LIN {X 0,Y 422.477,Z 421.748,A -85,B 0,C 180,E1 18512.668,E2 18512.668} C_VEL
LIN {X 0,Y 421.2,Z 421.073,A -85,B 0,C 180,E1 18507.876,E2 18507.876} C_VEL
LIN {X 0,Y 420.902,Z 420.888,A -85,B 0,C 180,E1 18503.227,E2 18503.227} C_VEL
LIN {X 0,Y 421.577,Z 421.279,A -85,B 0,C 180,E1 18498.545,E2 18498.545} C_VEL
LIN {X 0,Y 423.126,Z 422.074,A -85,B 0,C 180,E1 18494.007,E2 18494.007} C_VEL
LIN {X 0,Y 424.049,Z 423.451,A -85,B 0,C 180,E1 18491.958,E2 18491.958} C_VEL
LIN {X 0,Y 425.962,Z 426.546,A -85,B 0,C 180,E1 18488.466,E2 18488.466} C_VEL
LIN {X 0,Y 429.541,Z 429.118,A -85,B 0,C 180,E1 18484.205,E2 18484.205} C_VEL
LIN {X 0,Y 431.62,Z 432.69,A -85,B 0,C 180,E1 18481.882,E2 18481.882} C_VEL
LIN {X 0,Y 435.249,Z 435.605,A -85,B 0,C 180,E1 18478.844,E2 18478.844} C_VEL
LIN {X 0,Y 437.884,Z 439.562,A -85,B 0,C 180,E1 18476.733,E2 18476.733} C_VEL
LIN {X 0,Y 440.69,Z 442.015,A -85,B 0,C 180,E1 18474.818,E2 18474.818} C_VEL
LIN {X 0,Y 443.746,Z 446.143,A -85,B 0,C 180,E1 18472.838,E2 18472.838} C_VEL
LIN {X 0,Y 446.123,Z 448.296,A -85,B 0,C 180,E1 18471.471,E2 18471.471} C_VEL
LIN {X 0,Y 449.724,Z 452.865,A -85,B 0,C 180,E1 18469.489,E2 18469.489} C_VEL
LIN {X 0,Y 451.489,Z 454.777,A -85,B 0,C 180,E1 18468.581,E2 18468.581} C_VEL
LIN {X 0,Y 455.545,Z 459.465,A -85,B 0,C 180,E1 18466.645,E2 18466.645} C_VEL
LIN {X 0,Y 461.658,Z 466.953,A -85,B 0,C 180,E1 18463.946,E2 18463.946} C_VEL
LIN {X 0,Y 466.66,Z 473.171,A -85,B 0,C 180,E1 18461.933,E2 18461.933} C_VEL
LIN {X 0,Y 471.5,Z 479.208,A -85,B 0,C 180,E1 18460.138,E2 18460.138} C_VEL
LIN {X 0,Y 478.794,Z 488.277,A -85,B 0,C 180,E1 18457.651,E2 18457.651} C_VEL
LIN {X 0,Y 490.631,Z 503.832,A -85,B 0,C 180,E1 18454.032,E2 18454.032} C_VEL
LIN {X 0,Y 502.49,Z 520.193,A -85,B 0,C 180,E1 18450.827,E2 18450.827} C_VEL
LIN {X 0,Y 505.906,Z 525.431,A -85,B 0,C 180,E1 18449.952,E2 18449.952} C_VEL
LIN {X 0,Y 489.646,Z 725.558,A -85,B 0,C 180,E1 18446.587,E2 18446.587} C_VEL
LIN {X 0,Y 484.651,Z 786.492,A -85,B 0,C 180,E1 18445.522,E2 18445.522} C_VEL
LIN {X 0,Y 481.22,Z 813.949,A -85,B 0,C 180,E1 18444.851,E2 18444.851} C_VEL
LIN {X 0,Y 477.724,Z 836.513,A -85,B 0,C 180,E1 18444.155,E2 18444.155} C_VEL
LIN {X 0,Y 473.24,Z 860.935,A -85,B 0,C 180,E1 18443.241,E2 18443.241} C_VEL
LIN {X 0,Y 467.316,Z 887.73,A -85,B 0,C 180,E1 18442.006,E2 18442.006} C_VEL
LIN {X 0,Y 461.87,Z 909.342,A -85,B 0,C 180,E1 18440.819,E2 18440.819} C_VEL
LIN {X 0,Y 456.471,Z 928.774,A -85,B 0,C 180,E1 18439.587,E2 18439.587} C_VEL
LIN {X 0,Y 449.287,Z 952.388,A -85,B 0,C 180,E1 18437.86,E2 18437.86} C_VEL
LIN {X 0,Y 441.966,Z 973.956,A -85,B 0,C 180,E1 18435.991,E2 18435.991} C_VEL
LIN {X 0,Y 440.339,Z 978.566,A -85,B 0,C 180,E1 18435.558,E2 18435.558} C_VEL
LIN {X 0,Y 437.487,Z 984.737,A -85,B 0,C 180,E1 18435.064,E2 18435.064} C_VEL
LIN {X 0,Y 426.97,Z 1001.239,A -85,B 0,C 180,E1 18433.948,E2 18433.948} C_VEL
LIN {X 0,Y 424.489,Z 1006.084,A -85,B 0,C 180,E1 18433.45,E2 18433.45} C_VEL
LIN {X 0,Y 418.06,Z 1021.958,A -85,B 0,C 180,E1 18431.452,E2 18431.452} C_VEL
LIN {X 0,Y 411.031,Z 1038.717,A -85,B 0,C 180,E1 18429.048,E2 18429.048} C_VEL
LIN {X 0,Y 403.075,Z 1056.792,A -85,B 0,C 180,E1 18425.995,E2 18425.995} C_VEL
LIN {X 0,Y 397.406,Z 1069.465,A -85,B 0,C 180,E1 18423.513,E2 18423.513} C_VEL
LIN {X 0,Y 392.259,Z 1080.929,A -85,B 0,C 180,E1 18420.966,E2 18420.966} C_VEL
LIN {X 0,Y 387.642,Z 1091.318,A -85,B 0,C 180,E1 18418.344,E2 18418.344} C_VEL
LIN {X 0,Y 383.36,Z 1101.166,A -85,B 0,C 180,E1 18415.508,E2 18415.508} C_VEL
LIN {X 0,Y 378.871,Z 1112.052,A -85,B 0,C 180,E1 18411.856,E2 18411.856} C_VEL
LIN {X 0,Y 375.223,Z 1121.381,A -85,B 0,C 180,E1 18408.022,E2 18408.022} C_VEL
LIN {X 0,Y 372.964,Z 1127.882,A -85,B 0,C 180,E1 18404.837,E2 18404.837} C_VEL
LIN {X 0,Y 371.366,Z 1133.26,A -85,B 0,C 180,E1 18401.686,E2 18401.686} C_VEL
LIN {X 0,Y 370.296,Z 1137.459,A -85,B 0,C 180,E1 18398.707,E2 18398.707} C_VEL
LIN {X 0,Y 369.616,Z 1141.063,A -85,B 0,C 180,E1 18395.486,E2 18395.486} C_VEL
LIN {X 0,Y 369.252,Z 1143.784,A -85,B 0,C 180,E1 18392.239,E2 18392.239} C_VEL
LIN {X 0,Y 369.092,Z 1145.645,A -85,B 0,C 180,E1 18388.954,E2 18388.954} C_VEL
LIN {X 0,Y 369.086,Z 1146.802,A -85,B 0,C 180,E1 18385,E2 18385} C_VEL
LIN {X 0,Y 369.224,Z 1146.542,A -85,B 0,C 180,E1 18381.111,E2 18381.111} C_VEL
LIN {X 0,Y 369.509,Z 1145.383,A -85,B 0,C 180,E1 18377.732,E2 18377.732} C_VEL
LIN {X 0,Y 370.007,Z 1143.483,A -85,B 0,C 180,E1 18374.556,E2 18374.556} C_VEL
LIN {X 0,Y 370.928,Z 1140.504,A -85,B 0,C 180,E1 18371.128,E2 18371.128} C_VEL
LIN {X 0,Y 372.332,Z 1136.75,A -85,B 0,C 180,E1 18367.872,E2 18367.872} C_VEL
LIN {X 0,Y 375.08,Z 1130.512,A -85,B 0,C 180,E1 18363.668,E2 18363.668} C_VEL
LIN {X 0,Y 378.427,Z 1123.493,A -85,B 0,C 180,E1 18360,E2 18360} C_VEL
LIN {X 0,Y 382.175,Z 1116.307,A -85,B 0,C 180,E1 18356.85,E2 18356.85} C_VEL
LIN {X 0,Y 387.709,Z 1106.342,A -85,B 0,C 180,E1 18353.163,E2 18353.163} C_VEL
LIN {X 0,Y 394.48,Z 1094.18,A -85,B 0,C 180,E1 18349.485,E2 18349.485} C_VEL
LIN {X 0,Y 400.892,Z 1082.925,A -85,B 0,C 180,E1 18346.588,E2 18346.588} C_VEL
LIN {X 0,Y 409.517,Z 1067.682,A -85,B 0,C 180,E1 18343.255,E2 18343.255} C_VEL
LIN {X 0,Y 417.178,Z 1053.814,A -85,B 0,C 180,E1 18340.685,E2 18340.685} C_VEL
LIN {X 0,Y 426.442,Z 1036.933,A -85,B 0,C 180,E1 18337.966,E2 18337.966} C_VEL
LIN {X 0,Y 436.985,Z 1016.878,A -85,B 0,C 180,E1 18335.245,E2 18335.245} C_VEL
LIN {X 0,Y 448.675,Z 994.533,A -85,B 0,C 180,E1 18332.672,E2 18332.672} C_VEL
LIN {X 0,Y 462.163,Z 969.434,A -85,B 0,C 180,E1 18330.23,E2 18330.23} C_VEL
LIN {X 0,Y 466.813,Z 961.351,A -85,B 0,C 180,E1 18329.495,E2 18329.495} C_VEL
LIN {X 0,Y 455.272,Z 985.103,A -85,B 0,C 180,E1 18328.085,E2 18328.085} C_VEL
LIN {X 0,Y 443.229,Z 1013.929,A -85,B 0,C 180,E1 18326.116,E2 18326.116} C_VEL
LIN {X 0,Y 430.672,Z 1047.911,A -85,B 0,C 180,E1 18323.446,E2 18323.446} C_VEL
LIN {X 0,Y 420.191,Z 1078.59,A -85,B 0,C 180,E1 18320.656,E2 18320.656} C_VEL
LIN {X 0,Y 412.782,Z 1100.763,A -85,B 0,C 180,E1 18318.332,E2 18318.332} C_VEL
LIN {X 0,Y 406.522,Z 1119.645,A -85,B 0,C 180,E1 18316.109,E2 18316.109} C_VEL
LIN {X 0,Y 400.734,Z 1137.311,A -85,B 0,C 180,E1 18313.779,E2 18313.779} C_VEL
LIN {X 0,Y 395.31,Z 1154.058,A -85,B 0,C 180,E1 18311.303,E2 18311.303} C_VEL
LIN {X 0,Y 389.457,Z 1172.495,A -85,B 0,C 180,E1 18308.221,E2 18308.221} C_VEL
LIN {X 0,Y 384.02,Z 1190.224,A -85,B 0,C 180,E1 18304.765,E2 18304.765} C_VEL
LIN {X 0,Y 380.188,Z 1203.337,A -85,B 0,C 180,E1 18301.844,E2 18301.844} C_VEL
LIN {X 0,Y 377.038,Z 1215.184,A -85,B 0,C 180,E1 18298.859,E2 18298.859} C_VEL
LIN {X 0,Y 374.31,Z 1226.337,A -85,B 0,C 180,E1 18295.642,E2 18295.642} C_VEL
LIN {X 0,Y 372.26,Z 1235.988,A -85,B 0,C 180,E1 18292.421,E2 18292.421} C_VEL
LIN {X 0,Y 370.742,Z 1244.662,A -85,B 0,C 180,E1 18289.046,E2 18289.046} C_VEL
LIN {X 0,Y 369.633,Z 1253.129,A -85,B 0,C 180,E1 18285.045,E2 18285.045} C_VEL
LIN {X 0,Y 369.185,Z 1259.081,A -85,B 0,C 180,E1 18281.403,E2 18281.403} C_VEL
LIN {X 0,Y 369.039,Z 1263.015,A -85,B 0,C 180,E1 18278.256,E2 18278.256} C_VEL
LIN {X 0,Y 369.058,Z 1265.774,A -85,B 0,C 180,E1 18275.129,E2 18275.129} C_VEL
LIN {X 0,Y 369.071,Z 1267.308,A -85,B 0,C 180,E1 18272.174,E2 18272.174} C_VEL
LIN {X 0,Y 368.998,Z 1267.794,A -85,B 0,C 180,E1 18269.189,E2 18269.189} C_VEL
LIN {X 0,Y 368.957,Z 1267.269,A -85,B 0,C 180,E1 18266.271,E2 18266.271} C_VEL
LIN {X 0,Y 368.868,Z 1265.586,A -85,B 0,C 180,E1 18263.15,E2 18263.15} C_VEL
LIN {X 0,Y 368.867,Z 1262.604,A -85,B 0,C 180,E1 18259.852,E2 18259.852} C_VEL
LIN {X 0,Y 369.078,Z 1258.854,A -85,B 0,C 180,E1 18256.846,E2 18256.846} C_VEL
LIN {X 0,Y 369.642,Z 1253.793,A -85,B 0,C 180,E1 18253.661,E2 18253.661} C_VEL
LIN {X 0,Y 370.657,Z 1247.56,A -85,B 0,C 180,E1 18250.458,E2 18250.458} C_VEL
LIN {X 0,Y 372.231,Z 1240.14,A -85,B 0,C 180,E1 18247.244,E2 18247.244} C_VEL
LIN {X 0,Y 374.579,Z 1231.04,A -85,B 0,C 180,E1 18243.868,E2 18243.868} C_VEL
LIN {X 0,Y 378.591,Z 1217.755,A -85,B 0,C 180,E1 18239.706,E2 18239.706} C_VEL
LIN {X 0,Y 382.841,Z 1205.184,A -85,B 0,C 180,E1 18236.38,E2 18236.38} C_VEL
LIN {X 0,Y 387.175,Z 1193.056,A -85,B 0,C 180,E1 18233.561,E2 18233.561} C_VEL
LIN {X 0,Y 392.551,Z 1178.799,A -85,B 0,C 180,E1 18230.637,E2 18230.637} C_VEL
LIN {X 0,Y 400.146,Z 1159.204,A -85,B 0,C 180,E1 18227.182,E2 18227.182} C_VEL
LIN {X 0,Y 406.5,Z 1142.784,A -85,B 0,C 180,E1 18224.695,E2 18224.695} C_VEL
LIN {X 0,Y 412.773,Z 1126.506,A -85,B 0,C 180,E1 18222.52,E2 18222.52} C_VEL
LIN {X 0,Y 420.255,Z 1106.798,A -85,B 0,C 180,E1 18220.206,E2 18220.206} C_VEL
LIN {X 0,Y 428.742,Z 1083.312,A -85,B 0,C 180,E1 18217.858,E2 18217.858} C_VEL
LIN {X 0,Y 435.625,Z 1063.438,A -85,B 0,C 180,E1 18216.15,E2 18216.15} C_VEL
LIN {X 0,Y 442.024,Z 1043.926,A -85,B 0,C 180,E1 18214.689,E2 18214.689} C_VEL
LIN {X 0,Y 449.76,Z 1018.549,A -85,B 0,C 180,E1 18213.058,E2 18213.058} C_VEL
LIN {X 0,Y 456.374,Z 994.527,A -85,B 0,C 180,E1 18211.78,E2 18211.78} C_VEL
LIN {X 0,Y 461.859,Z 972.769,A -85,B 0,C 180,E1 18210.804,E2 18210.804} C_VEL
LIN {X 0,Y 467.539,Z 947.635,A -85,B 0,C 180,E1 18209.865,E2 18209.865} C_VEL
LIN {X 0,Y 472.907,Z 919.323,A -85,B 0,C 180,E1 18209.041,E2 18209.041} C_VEL
LIN {X 0,Y 476.53,Z 895.135,A -85,B 0,C 180,E1 18208.474,E2 18208.474} C_VEL
LIN {X 0,Y 479.514,Z 866.232,A -85,B 0,C 180,E1 18207.909,E2 18207.909} C_VEL
LIN {X 0,Y 496.179,Z 662.467,A -85,B 0,C 180,E1 18204.412,E2 18204.412} C_VEL
LIN {X 0,Y 505.804,Z 552.027,A -85,B 0,C 180,E1 18202.52,E2 18202.52} C_VEL
LIN {X 0,Y 495.363,Z 534.889,A -85,B 0,C 180,E1 18199.638,E2 18199.638} C_VEL
LIN {X 0,Y 484.943,Z 518.705,A -85,B 0,C 180,E1 18196.47,E2 18196.47} C_VEL
LIN {X 0,Y 475.423,Z 504.357,A -85,B 0,C 180,E1 18193.222,E2 18193.222} C_VEL
LIN {X 0,Y 467.105,Z 492.351,A -85,B 0,C 180,E1 18190.046,E2 18190.046} C_VEL
LIN {X 0,Y 461.3,Z 484.13,A -85,B 0,C 180,E1 18187.598,E2 18187.598} C_VEL
LIN {X 0,Y 455.063,Z 475.157,A -85,B 0,C 180,E1 18184.663,E2 18184.663} C_VEL
LIN {X 0,Y 449.645,Z 467.853,A -85,B 0,C 180,E1 18181.848,E2 18181.848} C_VEL
LIN {X 0,Y 446.334,Z 463.256,A -85,B 0,C 180,E1 18179.936,E2 18179.936} C_VEL
LIN {X 0,Y 442.559,Z 457.983,A -85,B 0,C 180,E1 18177.54,E2 18177.54} C_VEL
LIN {X 0,Y 438.72,Z 452.686,A -85,B 0,C 180,E1 18174.845,E2 18174.845} C_VEL
LIN {X 0,Y 435.455,Z 448.134,A -85,B 0,C 180,E1 18172.28,E2 18172.28} C_VEL
LIN {X 0,Y 431.5,Z 442.541,A -85,B 0,C 180,E1 18168.64,E2 18168.64} C_VEL
LIN {X 0,Y 430.232,Z 440.915,A -85,B 0,C 180,E1 18167.381,E2 18167.381} C_VEL
LIN {X 0,Y 427.667,Z 437.207,A -85,B 0,C 180,E1 18164.418,E2 18164.418} C_VEL
LIN {X 0,Y 426.822,Z 436.185,A -85,B 0,C 180,E1 18163.36,E2 18163.36} C_VEL
LIN {X 0,Y 423.806,Z 433.731,A -85,B 0,C 180,E1 18159.111,E2 18159.111} C_VEL
LIN {X 0,Y 421.826,Z 430.232,A -85,B 0,C 180,E1 18154.887,E2 18154.887} C_VEL
LIN {X 0,Y 420.441,Z 429.353,A -85,B 0,C 180,E1 18151.133,E2 18151.133} C_VEL
LIN {X 0,Y 419.493,Z 428.83,A -85,B 0,C 180,E1 18146.427,E2 18146.427} C_VEL
LIN {X 0,Y 419.54,Z 428.802,A -85,B 0,C 180,E1 18141.709,E2 18141.709} C_VEL
LIN {X 0,Y 420.481,Z 429.36,A -85,B 0,C 180,E1 18136.962,E2 18136.962} C_VEL
LIN {X 0,Y 422.003,Z 430.264,A -85,B 0,C 180,E1 18133.215,E2 18133.215} C_VEL
LIN {X 0,Y 424.327,Z 434.237,A -85,B 0,C 180,E1 18128.741,E2 18128.741} C_VEL
LIN {X 0,Y 427.943,Z 436.911,A -85,B 0,C 180,E1 18124.351,E2 18124.351} C_VEL
LIN {X 0,Y 430.109,Z 440.551,A -85,B 0,C 180,E1 18121.947,E2 18121.947} C_VEL
LIN {X 0,Y 433.609,Z 443.376,A -85,B 0,C 180,E1 18119.012,E2 18119.012} C_VEL
LIN {X 0,Y 436.28,Z 447.364,A -85,B 0,C 180,E1 18116.839,E2 18116.839} C_VEL
LIN {X 0,Y 439.009,Z 449.815,A -85,B 0,C 180,E1 18114.975,E2 18114.975} C_VEL
LIN {X 0,Y 442.263,Z 454.05,A -85,B 0,C 180,E1 18112.884,E2 18112.884} C_VEL
LIN {X 0,Y 444.364,Z 456.017,A -85,B 0,C 180,E1 18111.655,E2 18111.655} C_VEL
LIN {X 0,Y 448.022,Z 460.593,A -85,B 0,C 180,E1 18109.64,E2 18109.64} C_VEL
LIN {X 0,Y 449.691,Z 462.475,A -85,B 0,C 180,E1 18108.77,E2 18108.77} C_VEL
LIN {X 0,Y 453.841,Z 467.22,A -85,B 0,C 180,E1 18106.775,E2 18106.775} C_VEL
LIN {X 0,Y 459.85,Z 474.764,A -85,B 0,C 180,E1 18104.095,E2 18104.095} C_VEL
LIN {X 0,Y 464.488,Z 480.493,A -85,B 0,C 180,E1 18102.226,E2 18102.226} C_VEL
LIN {X 0,Y 469.597,Z 486.952,A -85,B 0,C 180,E1 18100.303,E2 18100.303} C_VEL
LIN {X 0,Y 476.774,Z 495.993,A -85,B 0,C 180,E1 18097.835,E2 18097.835} C_VEL
LIN {X 0,Y 488.194,Z 511.093,A -85,B 0,C 180,E1 18094.313,E2 18094.313} C_VEL
LIN {X 0,Y 500.319,Z 527.958,A -85,B 0,C 180,E1 18091.002,E2 18091.002} C_VEL
LIN {X 0,Y 501.547,Z 530.191,A -85,B 0,C 180,E1 18090.668,E2 18090.668} C_VEL
LIN {X 0,Y 484.769,Z 730.579,A -85,B 0,C 180,E1 18087.285,E2 18087.285} C_VEL
LIN {X 0,Y 479.89,Z 787.869,A -85,B 0,C 180,E1 18086.274,E2 18086.274} C_VEL
LIN {X 0,Y 476.377,Z 815.183,A -85,B 0,C 180,E1 18085.6,E2 18085.6} C_VEL
LIN {X 0,Y 472.71,Z 838.22,A -85,B 0,C 180,E1 18084.884,E2 18084.884} C_VEL
LIN {X 0,Y 467.619,Z 865.048,A -85,B 0,C 180,E1 18083.863,E2 18083.863} C_VEL
LIN {X 0,Y 461.903,Z 889.907,A -85,B 0,C 180,E1 18082.694,E2 18082.694} C_VEL
LIN {X 0,Y 456.642,Z 910.383,A -85,B 0,C 180,E1 18081.564,E2 18081.564} C_VEL
LIN {X 0,Y 451.001,Z 930.274,A -85,B 0,C 180,E1 18080.3,E2 18080.3} C_VEL
LIN {X 0,Y 443.622,Z 953.844,A -85,B 0,C 180,E1 18078.56,E2 18078.56} C_VEL
LIN {X 0,Y 436.41,Z 974.581,A -85,B 0,C 180,E1 18076.755,E2 18076.755} C_VEL
LIN {X 0,Y 430.039,Z 991.806,A -85,B 0,C 180,E1 18075.044,E2 18075.044} C_VEL
LIN {X 0,Y 424.489,Z 1006.084,A -85,B 0,C 180,E1 18073.45,E2 18073.45} C_VEL
LIN {X 0,Y 421.519,Z 1011.888,A -85,B 0,C 180,E1 18072.863,E2 18072.863} C_VEL
LIN {X 0,Y 410.746,Z 1027.262,A -85,B 0,C 180,E1 18071.508,E2 18071.508} C_VEL
LIN {X 0,Y 408.204,Z 1031.79,A -85,B 0,C 180,E1 18070.931,E2 18070.931} C_VEL
LIN {X 0,Y 401.358,Z 1047.233,A -85,B 0,C 180,E1 18068.518,E2 18068.518} C_VEL
LIN {X 0,Y 395.242,Z 1060.698,A -85,B 0,C 180,E1 18066.124,E2 18066.124} C_VEL
LIN {X 0,Y 389.422,Z 1073.347,A -85,B 0,C 180,E1 18063.554,E2 18063.554} C_VEL
LIN {X 0,Y 382.74,Z 1087.866,A -85,B 0,C 180,E1 18060.151,E2 18060.151} C_VEL
LIN {X 0,Y 377.037,Z 1100.262,A -85,B 0,C 180,E1 18056.655,E2 18056.655} C_VEL
LIN {X 0,Y 373.014,Z 1109.391,A -85,B 0,C 180,E1 18053.673,E2 18053.673} C_VEL
LIN {X 0,Y 369.711,Z 1117.344,A -85,B 0,C 180,E1 18050.669,E2 18050.669} C_VEL
LIN {X 0,Y 366.845,Z 1124.777,A -85,B 0,C 180,E1 18047.386,E2 18047.386} C_VEL
LIN {X 0,Y 364.262,Z 1132.422,A -85,B 0,C 180,E1 18043.331,E2 18043.331} C_VEL
LIN {X 0,Y 362.619,Z 1138.147,A -85,B 0,C 180,E1 18039.361,E2 18039.361} C_VEL
LIN {X 0,Y 361.821,Z 1141.9,A -85,B 0,C 180,E1 18036.06,E2 18036.06} C_VEL
LIN {X 0,Y 361.394,Z 1144.55,A -85,B 0,C 180,E1 18033.028,E2 18033.028} C_VEL
LIN {X 0,Y 361.226,Z 1146.499,A -85,B 0,C 180,E1 18029.884,E2 18029.884} C_VEL
LIN {X 0,Y 361.136,Z 1147.664,A -85,B 0,C 180,E1 18026.828,E2 18026.828} C_VEL
LIN {X 0,Y 361.215,Z 1148.095,A -85,B 0,C 180,E1 18023.665,E2 18023.665} C_VEL
LIN {X 0,Y 361.366,Z 1147.789,A -85,B 0,C 180,E1 18020.573,E2 18020.573} C_VEL
LIN {X 0,Y 361.689,Z 1146.695,A -85,B 0,C 180,E1 18017.372,E2 18017.372} C_VEL
LIN {X 0,Y 362.269,Z 1144.732,A -85,B 0,C 180,E1 18014.057,E2 18014.057} C_VEL
LIN {X 0,Y 363.285,Z 1141.804,A -85,B 0,C 180,E1 18010.627,E2 18010.627} C_VEL
LIN {X 0,Y 365.305,Z 1137.079,A -85,B 0,C 180,E1 18006.503,E2 18006.503} C_VEL
LIN {X 0,Y 368.386,Z 1130.54,A -85,B 0,C 180,E1 18002.333,E2 18002.333} C_VEL
LIN {X 0,Y 371.664,Z 1124.318,A -85,B 0,C 180,E1 17999.075,E2 17999.075} C_VEL
LIN {X 0,Y 376.367,Z 1115.997,A -85,B 0,C 180,E1 17995.429,E2 17995.429} C_VEL
LIN {X 0,Y 382.876,Z 1104.81,A -85,B 0,C 180,E1 17991.439,E2 17991.439} C_VEL
LIN {X 0,Y 388.892,Z 1094.764,A -85,B 0,C 180,E1 17988.431,E2 17988.431} C_VEL
LIN {X 0,Y 396.77,Z 1081.826,A -85,B 0,C 180,E1 17985.105,E2 17985.105} C_VEL
LIN {X 0,Y 405.581,Z 1066.833,A -85,B 0,C 180,E1 17981.903,E2 17981.903} C_VEL
LIN {X 0,Y 415.512,Z 1049.986,A -85,B 0,C 180,E1 17978.841,E2 17978.841} C_VEL
LIN {X 0,Y 425.482,Z 1032.481,A -85,B 0,C 180,E1 17976.159,E2 17976.159} C_VEL
LIN {X 0,Y 437.558,Z 1011.323,A -85,B 0,C 180,E1 17973.391,E2 17973.391} C_VEL
LIN {X 0,Y 450.513,Z 989.108,A -85,B 0,C 180,E1 17970.918,E2 17970.918} C_VEL
LIN {X 0,Y 458.124,Z 976.648,A -85,B 0,C 180,E1 17969.665,E2 17969.665} C_VEL
LIN {X 0,Y 446.197,Z 999.628,A -85,B 0,C 180,E1 17968.135,E2 17968.135} C_VEL
LIN {X 0,Y 432.914,Z 1029.777,A -85,B 0,C 180,E1 17965.858,E2 17965.858} C_VEL
LIN {X 0,Y 419.608,Z 1064.071,A -85,B 0,C 180,E1 17962.851,E2 17962.851} C_VEL
LIN {X 0,Y 408.885,Z 1093.844,A -85,B 0,C 180,E1 17959.834,E2 17959.834} C_VEL
LIN {X 0,Y 401.321,Z 1115.374,A -85,B 0,C 180,E1 17957.305,E2 17957.305} C_VEL
LIN {X 0,Y 394.881,Z 1133.98,A -85,B 0,C 180,E1 17954.846,E2 17954.846} C_VEL
LIN {X 0,Y 389.11,Z 1150.989,A -85,B 0,C 180,E1 17952.318,E2 17952.318} C_VEL
LIN {X 0,Y 383.48,Z 1167.9,A -85,B 0,C 180,E1 17949.484,E2 17949.484} C_VEL
LIN {X 0,Y 377.163,Z 1187.519,A -85,B 0,C 180,E1 17945.678,E2 17945.678} C_VEL
LIN {X 0,Y 372.997,Z 1201.179,A -85,B 0,C 180,E1 17942.603,E2 17942.603} C_VEL
LIN {X 0,Y 369.724,Z 1212.734,A -85,B 0,C 180,E1 17939.663,E2 17939.663} C_VEL
LIN {X 0,Y 366.965,Z 1223.536,A -85,B 0,C 180,E1 17936.542,E2 17936.542} C_VEL
LIN {X 0,Y 364.702,Z 1233.423,A -85,B 0,C 180,E1 17933.253,E2 17933.253} C_VEL
LIN {X 0,Y 363.096,Z 1241.887,A -85,B 0,C 180,E1 17929.966,E2 17929.966} C_VEL
LIN {X 0,Y 362.021,Z 1249.377,A -85,B 0,C 180,E1 17926.528,E2 17926.528} C_VEL
LIN {X 0,Y 361.336,Z 1256.532,A -85,B 0,C 180,E1 17922.465,E2 17922.465} C_VEL
LIN {X 0,Y 361.123,Z 1261.335,A -85,B 0,C 180,E1 17918.705,E2 17918.705} C_VEL
LIN {X 0,Y 361.154,Z 1264.302,A -85,B 0,C 180,E1 17915.401,E2 17915.401} C_VEL
LIN {X 0,Y 361.178,Z 1265.982,A -85,B 0,C 180,E1 17912.221,E2 17912.221} C_VEL
LIN {X 0,Y 361.104,Z 1266.499,A -85,B 0,C 180,E1 17909.207,E2 17909.207} C_VEL
LIN {X 0,Y 361.054,Z 1265.982,A -85,B 0,C 180,E1 17906.189,E2 17906.189} C_VEL
LIN {X 0,Y 360.951,Z 1264.3,A -85,B 0,C 180,E1 17902.999,E2 17902.999} C_VEL
LIN {X 0,Y 360.95,Z 1261.304,A -85,B 0,C 180,E1 17899.627,E2 17899.627} C_VEL
LIN {X 0,Y 361.166,Z 1257.529,A -85,B 0,C 180,E1 17896.553,E2 17896.553} C_VEL
LIN {X 0,Y 361.761,Z 1252.434,A -85,B 0,C 180,E1 17893.295,E2 17893.295} C_VEL
LIN {X 0,Y 362.833,Z 1246.149,A -85,B 0,C 180,E1 17890.006,E2 17890.006} C_VEL
LIN {X 0,Y 364.504,Z 1238.734,A -85,B 0,C 180,E1 17886.733,E2 17886.733} C_VEL
LIN {X 0,Y 367.143,Z 1229.146,A -85,B 0,C 180,E1 17883.123,E2 17883.123} C_VEL
LIN {X 0,Y 371.24,Z 1216.193,A -85,B 0,C 180,E1 17879.041,E2 17879.041} C_VEL
LIN {X 0,Y 375.46,Z 1204.193,A -85,B 0,C 180,E1 17875.812,E2 17875.812} C_VEL
LIN {X 0,Y 380.151,Z 1191.626,A -85,B 0,C 180,E1 17872.841,E2 17872.841} C_VEL
LIN {X 0,Y 385.888,Z 1177.064,A -85,B 0,C 180,E1 17869.82,E2 17869.82} C_VEL
LIN {X 0,Y 393.651,Z 1157.614,A -85,B 0,C 180,E1 17866.379,E2 17866.379} C_VEL
LIN {X 0,Y 400.278,Z 1141.051,A -85,B 0,C 180,E1 17863.852,E2 17863.852} C_VEL
LIN {X 0,Y 407.473,Z 1123.005,A -85,B 0,C 180,E1 17861.44,E2 17861.44} C_VEL
LIN {X 0,Y 416.602,Z 1099.353,A -85,B 0,C 180,E1 17858.737,E2 17858.737} C_VEL
LIN {X 0,Y 423.689,Z 1080.141,A -85,B 0,C 180,E1 17856.868,E2 17856.868} C_VEL
LIN {X 0,Y 430.664,Z 1060.388,A -85,B 0,C 180,E1 17855.191,E2 17855.191} C_VEL
LIN {X 0,Y 438.973,Z 1035.382,A -85,B 0,C 180,E1 17853.368,E2 17853.368} C_VEL
LIN {X 0,Y 446.121,Z 1011.773,A -85,B 0,C 180,E1 17851.934,E2 17851.934} C_VEL
LIN {X 0,Y 452.241,Z 989.836,A -85,B 0,C 180,E1 17850.801,E2 17850.801} C_VEL
LIN {X 0,Y 459.038,Z 962.957,A -85,B 0,C 180,E1 17849.646,E2 17849.646} C_VEL
LIN {X 0,Y 464.732,Z 936.465,A -85,B 0,C 180,E1 17848.748,E2 17848.748} C_VEL
LIN {X 0,Y 469.047,Z 913.166,A -85,B 0,C 180,E1 17848.117,E2 17848.117} C_VEL
LIN {X 0,Y 473.049,Z 884.759,A -85,B 0,C 180,E1 17847.474,E2 17847.474} C_VEL
LIN {X 0,Y 478.086,Z 826.315,A -85,B 0,C 180,E1 17846.434,E2 17846.434} C_VEL
LIN {X 0,Y 496.063,Z 616.45,A -85,B 0,C 180,E1 17842.832,E2 17842.832} C_VEL
LIN {X 0,Y 501.431,Z 556.448,A -85,B 0,C 180,E1 17841.802,E2 17841.802} C_VEL
LIN {X 0,Y 491.609,Z 540.321,A -85,B 0,C 180,E1 17839.022,E2 17839.022} C_VEL
LIN {X 0,Y 482.063,Z 525.326,A -85,B 0,C 180,E1 17836.045,E2 17836.045} C_VEL
LIN {X 0,Y 473.136,Z 511.676,A -85,B 0,C 180,E1 17832.945,E2 17832.945} C_VEL
LIN {X 0,Y 465.089,Z 499.976,A -85,B 0,C 180,E1 17829.841,E2 17829.841} C_VEL
LIN {X 0,Y 459.222,Z 491.521,A -85,B 0,C 180,E1 17827.318,E2 17827.318} C_VEL
LIN {X 0,Y 453.016,Z 482.555,A -85,B 0,C 180,E1 17824.367,E2 17824.367} C_VEL
LIN {X 0,Y 447.744,Z 475.378,A -85,B 0,C 180,E1 17821.6,E2 17821.6} C_VEL
LIN {X 0,Y 444.415,Z 470.773,A -85,B 0,C 180,E1 17819.678,E2 17819.678} C_VEL
LIN {X 0,Y 440.749,Z 465.616,A -85,B 0,C 180,E1 17817.334,E2 17817.334} C_VEL
LIN {X 0,Y 436.935,Z 460.315,A -85,B 0,C 180,E1 17814.616,E2 17814.616} C_VEL
LIN {X 0,Y 433.641,Z 455.597,A -85,B 0,C 180,E1 17811.981,E2 17811.981} C_VEL
LIN {X 0,Y 429.892,Z 450.387,A -85,B 0,C 180,E1 17808.529,E2 17808.529} C_VEL
LIN {X 0,Y 428.839,Z 448.916,A -85,B 0,C 180,E1 17807.476,E2 17807.476} C_VEL
LIN {X 0,Y 426.205,Z 445.308,A -85,B 0,C 180,E1 17804.487,E2 17804.487} C_VEL
LIN {X 0,Y 425.435,Z 444.11,A -85,B 0,C 180,E1 17803.478,E2 17803.478} C_VEL
LIN {X 0,Y 422.356,Z 441.674,A -85,B 0,C 180,E1 17799.2,E2 17799.2} C_VEL
LIN {X 0,Y 420.543,Z 438.38,A -85,B 0,C 180,E1 17795.412,E2 17795.412} C_VEL
LIN {X 0,Y 419.286,Z 437.397,A -85,B 0,C 180,E1 17792.288,E2 17792.288} C_VEL
LIN {X 0,Y 418.174,Z 436.775,A -85,B 0,C 180,E1 17787.777,E2 17787.777} C_VEL
LIN {X 0,Y 417.876,Z 436.598,A -85,B 0,C 180,E1 17783.259,E2 17783.259} C_VEL
LIN {X 0,Y 418.501,Z 436.962,A -85,B 0,C 180,E1 17778.815,E2 17778.815} C_VEL
LIN {X 0,Y 420.06,Z 437.739,A -85,B 0,C 180,E1 17774.221,E2 17774.221} C_VEL
LIN {X 0,Y 420.983,Z 439.026,A -85,B 0,C 180,E1 17772.233,E2 17772.233} C_VEL
LIN {X 0,Y 423.002,Z 442.287,A -85,B 0,C 180,E1 17768.517,E2 17768.517} C_VEL
LIN {X 0,Y 426.348,Z 444.702,A -85,B 0,C 180,E1 17764.497,E2 17764.497} C_VEL
LIN {X 0,Y 428.638,Z 448.459,A -85,B 0,C 180,E1 17761.973,E2 17761.973} C_VEL
LIN {X 0,Y 431.985,Z 451.176,A -85,B 0,C 180,E1 17759.166,E2 17759.166} C_VEL
LIN {X 0,Y 434.674,Z 455.166,A -85,B 0,C 180,E1 17756.946,E2 17756.946} C_VEL
LIN {X 0,Y 437.283,Z 457.514,A -85,B 0,C 180,E1 17755.17,E2 17755.17} C_VEL
LIN {X 0,Y 440.553,Z 461.761,A -85,B 0,C 180,E1 17753.048,E2 17753.048} C_VEL
LIN {X 0,Y 442.653,Z 463.807,A -85,B 0,C 180,E1 17751.814,E2 17751.814} C_VEL
LIN {X 0,Y 446.488,Z 468.488,A -85,B 0,C 180,E1 17749.696,E2 17749.696} C_VEL
LIN {X 0,Y 448.182,Z 470.593,A -85,B 0,C 180,E1 17748.807,E2 17748.807} C_VEL
LIN {X 0,Y 452.937,Z 476.216,A -85,B 0,C 180,E1 17746.512,E2 17746.512} C_VEL
LIN {X 0,Y 457.714,Z 482.108,A -85,B 0,C 180,E1 17744.388,E2 17744.388} C_VEL
LIN {X 0,Y 462.717,Z 488.376,A -85,B 0,C 180,E1 17742.353,E2 17742.353} C_VEL
LIN {X 0,Y 469.919,Z 497.371,A -85,B 0,C 180,E1 17739.677,E2 17739.677} C_VEL
LIN {X 0,Y 478.554,Z 508.779,A -85,B 0,C 180,E1 17736.78,E2 17736.78} C_VEL
LIN {X 0,Y 488.748,Z 522.481,A -85,B 0,C 180,E1 17733.724,E2 17733.724} C_VEL
LIN {X 0,Y 497.273,Z 534.683,A -85,B 0,C 180,E1 17731.399,E2 17731.399} C_VEL
LIN {X 0,Y 479.238,Z 743.965,A -85,B 0,C 180,E1 17727.851,E2 17727.851} C_VEL
LIN {X 0,Y 475.149,Z 789.706,A -85,B 0,C 180,E1 17727.03,E2 17727.03} C_VEL
LIN {X 0,Y 471.621,Z 816.372,A -85,B 0,C 180,E1 17726.366,E2 17726.366} C_VEL
LIN {X 0,Y 467.872,Z 839.318,A -85,B 0,C 180,E1 17725.649,E2 17725.649} C_VEL
LIN {X 0,Y 462.725,Z 865.824,A -85,B 0,C 180,E1 17724.638,E2 17724.638} C_VEL
LIN {X 0,Y 456.708,Z 891.36,A -85,B 0,C 180,E1 17723.432,E2 17723.432} C_VEL
LIN {X 0,Y 451.324,Z 911.789,A -85,B 0,C 180,E1 17722.297,E2 17722.297} C_VEL
LIN {X 0,Y 445.437,Z 932.047,A -85,B 0,C 180,E1 17721.001,E2 17721.001} C_VEL
LIN {X 0,Y 437.371,Z 957.042,A -85,B 0,C 180,E1 17719.129,E2 17719.129} C_VEL
LIN {X 0,Y 430.632,Z 976.028,A -85,B 0,C 180,E1 17717.462,E2 17717.462} C_VEL
LIN {X 0,Y 424.051,Z 993.351,A -85,B 0,C 180,E1 17715.725,E2 17715.725} C_VEL
LIN {X 0,Y 416.986,Z 1011.002,A -85,B 0,C 180,E1 17713.707,E2 17713.707} C_VEL
LIN {X 0,Y 408.204,Z 1031.79,A -85,B 0,C 180,E1 17710.931,E2 17710.931} C_VEL
LIN {X 0,Y 405.144,Z 1037.079,A -85,B 0,C 180,E1 17710.246,E2 17710.246} C_VEL
LIN {X 0,Y 394.177,Z 1051.335,A -85,B 0,C 180,E1 17708.626,E2 17708.626} C_VEL
LIN {X 0,Y 391.683,Z 1055.538,A -85,B 0,C 180,E1 17707.974,E2 17707.974} C_VEL
LIN {X 0,Y 384.095,Z 1071.421,A -85,B 0,C 180,E1 17704.848,E2 17704.848} C_VEL
LIN {X 0,Y 378.344,Z 1083.477,A -85,B 0,C 180,E1 17702.11,E2 17702.11} C_VEL
LIN {X 0,Y 373.243,Z 1094.229,A -85,B 0,C 180,E1 17699.31,E2 17699.31} C_VEL
LIN {X 0,Y 367.77,Z 1106.06,A -85,B 0,C 180,E1 17695.743,E2 17695.743} C_VEL
LIN {X 0,Y 362.895,Z 1116.971,A -85,B 0,C 180,E1 17691.746,E2 17691.746} C_VEL
LIN {X 0,Y 359.902,Z 1124.226,A -85,B 0,C 180,E1 17688.601,E2 17688.601} C_VEL
LIN {X 0,Y 357.557,Z 1130.477,A -85,B 0,C 180,E1 17685.421,E2 17685.421} C_VEL
LIN {X 0,Y 355.735,Z 1136.103,A -85,B 0,C 180,E1 17681.987,E2 17681.987} C_VEL
LIN {X 0,Y 354.512,Z 1140.582,A -85,B 0,C 180,E1 17678.624,E2 17678.624} C_VEL
LIN {X 0,Y 353.697,Z 1144.958,A -85,B 0,C 180,E1 17674.365,E2 17674.365} C_VEL
LIN {X 0,Y 353.352,Z 1147.644,A -85,B 0,C 180,E1 17670.245,E2 17670.245} C_VEL
LIN {X 0,Y 353.242,Z 1148.955,A -85,B 0,C 180,E1 17666.922,E2 17666.922} C_VEL
LIN {X 0,Y 353.329,Z 1149.438,A -85,B 0,C 180,E1 17663.694,E2 17663.694} C_VEL
LIN {X 0,Y 353.491,Z 1149.178,A -85,B 0,C 180,E1 17660.533,E2 17660.533} C_VEL
LIN {X 0,Y 353.843,Z 1148.121,A -85,B 0,C 180,E1 17657.233,E2 17657.233} C_VEL
LIN {X 0,Y 354.462,Z 1146.236,A -85,B 0,C 180,E1 17653.873,E2 17653.873} C_VEL
LIN {X 0,Y 355.633,Z 1143.211,A -85,B 0,C 180,E1 17650.203,E2 17650.203} C_VEL
LIN {X 0,Y 357.869,Z 1138.415,A -85,B 0,C 180,E1 17645.929,E2 17645.929} C_VEL
LIN {X 0,Y 361.123,Z 1132.029,A -85,B 0,C 180,E1 17641.753,E2 17641.753} C_VEL
LIN {X 0,Y 364.823,Z 1125.502,A -85,B 0,C 180,E1 17638.272,E2 17638.272} C_VEL
LIN {X 0,Y 370.335,Z 1116.432,A -85,B 0,C 180,E1 17634.267,E2 17634.267} C_VEL
LIN {X 0,Y 376.493,Z 1106.411,A -85,B 0,C 180,E1 17630.677,E2 17630.677} C_VEL
LIN {X 0,Y 382.852,Z 1096.411,A -85,B 0,C 180,E1 17627.622,E2 17627.622} C_VEL
LIN {X 0,Y 391.084,Z 1083.596,A -85,B 0,C 180,E1 17624.275,E2 17624.275} C_VEL
LIN {X 0,Y 400.334,Z 1068.796,A -85,B 0,C 180,E1 17621.053,E2 17621.053} C_VEL
LIN {X 0,Y 411.187,Z 1051.437,A -85,B 0,C 180,E1 17617.857,E2 17617.857} C_VEL
LIN {X 0,Y 422.538,Z 1033.026,A -85,B 0,C 180,E1 17615.001,E2 17615.001} C_VEL
LIN {X 0,Y 436.765,Z 1010.158,A -85,B 0,C 180,E1 17612.01,E2 17612.01} C_VEL
LIN {X 0,Y 449.413,Z 990.847,A -85,B 0,C 180,E1 17609.831,E2 17609.831} C_VEL
LIN {X 0,Y 435.784,Z 1015.838,A -85,B 0,C 180,E1 17607.972,E2 17607.972} C_VEL
LIN {X 0,Y 423.14,Z 1043.176,A -85,B 0,C 180,E1 17605.676,E2 17605.676} C_VEL
LIN {X 0,Y 409.062,Z 1077.606,A -85,B 0,C 180,E1 17602.369,E2 17602.369} C_VEL
LIN {X 0,Y 398.279,Z 1106.302,A -85,B 0,C 180,E1 17599.16,E2 17599.16} C_VEL
LIN {X 0,Y 389.709,Z 1129.432,A -85,B 0,C 180,E1 17596.134,E2 17596.134} C_VEL
LIN {X 0,Y 383.717,Z 1146.078,A -85,B 0,C 180,E1 17593.672,E2 17593.672} C_VEL
LIN {X 0,Y 378.303,Z 1161.459,A -85,B 0,C 180,E1 17591.124,E2 17591.124} C_VEL
LIN {X 0,Y 373.32,Z 1176.038,A -85,B 0,C 180,E1 17588.416,E2 17588.416} C_VEL
LIN {X 0,Y 368.833,Z 1189.62,A -85,B 0,C 180,E1 17585.581,E2 17585.581} C_VEL
LIN {X 0,Y 364.924,Z 1202.007,A -85,B 0,C 180,E1 17582.668,E2 17582.668} C_VEL
LIN {X 0,Y 361.631,Z 1213.312,A -85,B 0,C 180,E1 17579.664,E2 17579.664} C_VEL
LIN {X 0,Y 358.72,Z 1224.451,A -85,B 0,C 180,E1 17576.307,E2 17576.307} C_VEL
LIN {X 0,Y 356.073,Z 1236.319,A -85,B 0,C 180,E1 17572.077,E2 17572.077} C_VEL
LIN {X 0,Y 354.496,Z 1245.149,A -85,B 0,C 180,E1 17568.245,E2 17568.245} C_VEL
LIN {X 0,Y 353.716,Z 1251.494,A -85,B 0,C 180,E1 17564.906,E2 17564.906} C_VEL
LIN {X 0,Y 353.366,Z 1256.413,A -85,B 0,C 180,E1 17561.749,E2 17561.749} C_VEL
LIN {X 0,Y 353.212,Z 1260.214,A -85,B 0,C 180,E1 17558.629,E2 17558.629} C_VEL
LIN {X 0,Y 353.253,Z 1262.942,A -85,B 0,C 180,E1 17555.522,E2 17555.522} C_VEL
LIN {X 0,Y 353.287,Z 1264.596,A -85,B 0,C 180,E1 17552.433,E2 17552.433} C_VEL
LIN {X 0,Y 353.214,Z 1265.189,A -85,B 0,C 180,E1 17549.351,E2 17549.351} C_VEL
LIN {X 0,Y 353.153,Z 1264.671,A -85,B 0,C 180,E1 17546.104,E2 17546.104} C_VEL
LIN {X 0,Y 353.029,Z 1262.987,A -85,B 0,C 180,E1 17542.841,E2 17542.841} C_VEL
LIN {X 0,Y 353.024,Z 1260.16,A -85,B 0,C 180,E1 17539.556,E2 17539.556} C_VEL
LIN {X 0,Y 353.231,Z 1256.423,A -85,B 0,C 180,E1 17536.412,E2 17536.412} C_VEL
LIN {X 0,Y 353.848,Z 1251.369,A -85,B 0,C 180,E1 17533.079,E2 17533.079} C_VEL
LIN {X 0,Y 354.947,Z 1245.143,A -85,B 0,C 180,E1 17529.727,E2 17529.727} C_VEL
LIN {X 0,Y 356.595,Z 1238.106,A -85,B 0,C 180,E1 17526.537,E2 17526.537} C_VEL
LIN {X 0,Y 359.026,Z 1229.479,A -85,B 0,C 180,E1 17523.182,E2 17523.182} C_VEL
LIN {X 0,Y 362.95,Z 1217.483,A -85,B 0,C 180,E1 17519.176,E2 17519.176} C_VEL
LIN {X 0,Y 367.878,Z 1203.849,A -85,B 0,C 180,E1 17515.385,E2 17515.385} C_VEL
LIN {X 0,Y 372.541,Z 1191.797,A -85,B 0,C 180,E1 17512.464,E2 17512.464} C_VEL
LIN {X 0,Y 377.981,Z 1178.36,A -85,B 0,C 180,E1 17509.601,E2 17509.601} C_VEL
LIN {X 0,Y 385.286,Z 1160.865,A -85,B 0,C 180,E1 17506.345,E2 17506.345} C_VEL
LIN {X 0,Y 393.157,Z 1141.744,A -85,B 0,C 180,E1 17503.335,E2 17503.335} C_VEL
LIN {X 0,Y 399.749,Z 1125.732,A -85,B 0,C 180,E1 17501.136,E2 17501.136} C_VEL
LIN {X 0,Y 406.759,Z 1108.31,A -85,B 0,C 180,E1 17499.034,E2 17499.034} C_VEL
LIN {X 0,Y 415.362,Z 1086.214,A -85,B 0,C 180,E1 17496.716,E2 17496.716} C_VEL
LIN {X 0,Y 423.481,Z 1063.966,A -85,B 0,C 180,E1 17494.749,E2 17494.749} C_VEL
LIN {X 0,Y 430.356,Z 1044.188,A -85,B 0,C 180,E1 17493.237,E2 17493.237} C_VEL
LIN {X 0,Y 437.518,Z 1022.109,A -85,B 0,C 180,E1 17491.773,E2 17491.773} C_VEL
LIN {X 0,Y 445.664,Z 994.531,A -85,B 0,C 180,E1 17490.257,E2 17490.257} C_VEL
LIN {X 0,Y 451.375,Z 973.032,A -85,B 0,C 180,E1 17489.282,E2 17489.282} C_VEL
LIN {X 0,Y 456.587,Z 951.211,A -85,B 0,C 180,E1 17488.449,E2 17488.449} C_VEL
LIN {X 0,Y 462.3,Z 924.041,A -85,B 0,C 180,E1 17487.607,E2 17487.607} C_VEL
LIN {X 0,Y 466.723,Z 896.752,A -85,B 0,C 180,E1 17486.949,E2 17486.949} C_VEL
LIN {X 0,Y 469.431,Z 873.652,A -85,B 0,C 180,E1 17486.476,E2 17486.476} C_VEL
LIN {X 0,Y 489.134,Z 648.142,A -85,B 0,C 180,E1 17482.569,E2 17482.569} C_VEL
LIN {X 0,Y 497.209,Z 560.98,A -85,B 0,C 180,E1 17481.071,E2 17481.071} C_VEL
LIN {X 0,Y 488.24,Z 546.178,A -85,B 0,C 180,E1 17478.477,E2 17478.477} C_VEL
LIN {X 0,Y 479.306,Z 532.071,A -85,B 0,C 180,E1 17475.642,E2 17475.642} C_VEL
LIN {X 0,Y 470.853,Z 518.996,A -85,B 0,C 180,E1 17472.666,E2 17472.666} C_VEL
LIN {X 0,Y 462.784,Z 507.164,A -85,B 0,C 180,E1 17469.514,E2 17469.514} C_VEL
LIN {X 0,Y 457.098,Z 498.898,A -85,B 0,C 180,E1 17467.036,E2 17467.036} C_VEL
LIN {X 0,Y 450.951,Z 489.943,A -85,B 0,C 180,E1 17464.069,E2 17464.069} C_VEL
LIN {X 0,Y 445.851,Z 482.903,A -85,B 0,C 180,E1 17461.349,E2 17461.349} C_VEL
LIN {X 0,Y 442.397,Z 478.158,A -85,B 0,C 180,E1 17459.352,E2 17459.352} C_VEL
LIN {X 0,Y 438.84,Z 473.131,A -85,B 0,C 180,E1 17457.061,E2 17457.061} C_VEL
LIN {X 0,Y 435.244,Z 468.046,A -85,B 0,C 180,E1 17454.463,E2 17454.463} C_VEL
LIN {X 0,Y 431.905,Z 463.206,A -85,B 0,C 180,E1 17451.748,E2 17451.748} C_VEL
LIN {X 0,Y 428.223,Z 458.099,A -85,B 0,C 180,E1 17448.347,E2 17448.347} C_VEL
LIN {X 0,Y 427.157,Z 456.632,A -85,B 0,C 180,E1 17447.289,E2 17447.289} C_VEL
LIN {X 0,Y 424.616,Z 453.143,A -85,B 0,C 180,E1 17444.387,E2 17444.387} C_VEL
LIN {X 0,Y 423.809,Z 451.897,A -85,B 0,C 180,E1 17443.307,E2 17443.307} C_VEL
LIN {X 0,Y 420.747,Z 449.452,A -85,B 0,C 180,E1 17439.057,E2 17439.057} C_VEL
LIN {X 0,Y 419.01,Z 446.28,A -85,B 0,C 180,E1 17435.391,E2 17435.391} C_VEL
LIN {X 0,Y 417.852,Z 445.286,A -85,B 0,C 180,E1 17432.494,E2 17432.494} C_VEL
LIN {X 0,Y 416.673,Z 444.638,A -85,B 0,C 180,E1 17427.809,E2 17427.809} C_VEL
LIN {X 0,Y 416.364,Z 444.452,A -85,B 0,C 180,E1 17423.275,E2 17423.275} C_VEL
LIN {X 0,Y 416.92,Z 444.786,A -85,B 0,C 180,E1 17419.064,E2 17419.064} C_VEL
LIN {X 0,Y 418.572,Z 445.602,A -85,B 0,C 180,E1 17414.222,E2 17414.222} C_VEL
LIN {X 0,Y 419.42,Z 446.829,A -85,B 0,C 180,E1 17412.35,E2 17412.35} C_VEL
LIN {X 0,Y 421.484,Z 450.116,A -85,B 0,C 180,E1 17408.602,E2 17408.602} C_VEL
LIN {X 0,Y 424.754,Z 452.494,A -85,B 0,C 180,E1 17404.645,E2 17404.645} C_VEL
LIN {X 0,Y 427.099,Z 456.289,A -85,B 0,C 180,E1 17402.06,E2 17402.06} C_VEL
LIN {X 0,Y 430.306,Z 458.881,A -85,B 0,C 180,E1 17399.36,E2 17399.36} C_VEL
LIN {X 0,Y 433.154,Z 463.05,A -85,B 0,C 180,E1 17396.995,E2 17396.995} C_VEL
LIN {X 0,Y 435.597,Z 465.275,A -85,B 0,C 180,E1 17395.339,E2 17395.339} C_VEL
LIN {X 0,Y 439.081,Z 469.691,A -85,B 0,C 180,E1 17393.073,E2 17393.073} C_VEL
LIN {X 0,Y 440.832,Z 471.396,A -85,B 0,C 180,E1 17392.048,E2 17392.048} C_VEL
LIN {X 0,Y 444.778,Z 476.22,A -85,B 0,C 180,E1 17389.844,E2 17389.844} C_VEL
LIN {X 0,Y 450.986,Z 483.752,A -85,B 0,C 180,E1 17386.752,E2 17386.752} C_VEL
LIN {X 0,Y 455.75,Z 489.676,A -85,B 0,C 180,E1 17384.614,E2 17384.614} C_VEL
LIN {X 0,Y 460.716,Z 495.959,A -85,B 0,C 180,E1 17382.566,E2 17382.566} C_VEL
LIN {X 0,Y 467.636,Z 504.652,A -85,B 0,C 180,E1 17379.973,E2 17379.973} C_VEL
LIN {X 0,Y 476.334,Z 516.236,A -85,B 0,C 180,E1 17377.023,E2 17377.023} C_VEL
LIN {X 0,Y 486.387,Z 529.882,A -85,B 0,C 180,E1 17373.978,E2 17373.978} C_VEL
LIN {X 0,Y 492.952,Z 539.538,A -85,B 0,C 180,E1 17372.131,E2 17372.131} C_VEL
LIN {X 0,Y 474.716,Z 745.837,A -85,B 0,C 180,E1 17368.627,E2 17368.627} C_VEL
LIN {X 0,Y 470.52,Z 791.097,A -85,B 0,C 180,E1 17367.808,E2 17367.808} C_VEL
LIN {X 0,Y 466.967,Z 817.351,A -85,B 0,C 180,E1 17367.152,E2 17367.152} C_VEL
LIN {X 0,Y 463.245,Z 839.708,A -85,B 0,C 180,E1 17366.454,E2 17366.454} C_VEL
LIN {X 0,Y 458.084,Z 865.809,A -85,B 0,C 180,E1 17365.462,E2 17365.462} C_VEL
LIN {X 0,Y 451.934,Z 891.492,A -85,B 0,C 180,E1 17364.254,E2 17364.254} C_VEL
LIN {X 0,Y 446.21,Z 912.746,A -85,B 0,C 180,E1 17363.074,E2 17363.074} C_VEL
LIN {X 0,Y 440.173,Z 933.034,A -85,B 0,C 180,E1 17361.772,E2 17361.772} C_VEL
LIN {X 0,Y 431.786,Z 958.371,A -85,B 0,C 180,E1 17359.864,E2 17359.864} C_VEL
LIN {X 0,Y 424.883,Z 977.357,A -85,B 0,C 180,E1 17358.186,E2 17358.186} C_VEL
LIN {X 0,Y 418.193,Z 994.62,A -85,B 0,C 180,E1 17356.449,E2 17356.449} C_VEL
LIN {X 0,Y 411.028,Z 1012.141,A -85,B 0,C 180,E1 17354.437,E2 17354.437} C_VEL
LIN {X 0,Y 401.812,Z 1033.314,A -85,B 0,C 180,E1 17351.577,E2 17351.577} C_VEL
LIN {X 0,Y 395.079,Z 1048.078,A -85,B 0,C 180,E1 17349.249,E2 17349.249} C_VEL
LIN {X 0,Y 391.683,Z 1055.538,A -85,B 0,C 180,E1 17347.974,E2 17347.974} C_VEL
LIN {X 0,Y 388.676,Z 1060.378,A -85,B 0,C 180,E1 17347.199,E2 17347.199} C_VEL
LIN {X 0,Y 377.676,Z 1073.21,A -85,B 0,C 180,E1 17345.275,E2 17345.275} C_VEL
LIN {X 0,Y 375.265,Z 1077.011,A -85,B 0,C 180,E1 17344.53,E2 17344.53} C_VEL
LIN {X 0,Y 367.755,Z 1092.195,A -85,B 0,C 180,E1 17340.783,E2 17340.783} C_VEL
LIN {X 0,Y 362.543,Z 1102.909,A -85,B 0,C 180,E1 17337.653,E2 17337.653} C_VEL
LIN {X 0,Y 358.254,Z 1111.997,A -85,B 0,C 180,E1 17334.585,E2 17334.585} C_VEL
LIN {X 0,Y 354.428,Z 1120.531,A -85,B 0,C 180,E1 17331.224,E2 17331.224} C_VEL
LIN {X 0,Y 350.827,Z 1129.406,A -85,B 0,C 180,E1 17327.066,E2 17327.066} C_VEL
LIN {X 0,Y 348.269,Z 1136.337,A -85,B 0,C 180,E1 17322.937,E2 17322.937} C_VEL
LIN {X 0,Y 346.915,Z 1140.934,A -85,B 0,C 180,E1 17319.567,E2 17319.567} C_VEL
LIN {X 0,Y 346.088,Z 1144.51,A -85,B 0,C 180,E1 17316.288,E2 17316.288} C_VEL
LIN {X 0,Y 345.623,Z 1147.156,A -85,B 0,C 180,E1 17313.147,E2 17313.147} C_VEL
LIN {X 0,Y 345.437,Z 1149.127,A -85,B 0,C 180,E1 17309.859,E2 17309.859} C_VEL
LIN {X 0,Y 345.359,Z 1150.311,A -85,B 0,C 180,E1 17306.664,E2 17306.664} C_VEL
LIN {X 0,Y 345.439,Z 1150.769,A -85,B 0,C 180,E1 17303.544,E2 17303.544} C_VEL
LIN {X 0,Y 345.63,Z 1150.526,A -85,B 0,C 180,E1 17300.314,E2 17300.314} C_VEL
LIN {X 0,Y 346.015,Z 1149.51,A -85,B 0,C 180,E1 17296.965,E2 17296.965} C_VEL
LIN {X 0,Y 346.697,Z 1147.638,A -85,B 0,C 180,E1 17293.51,E2 17293.51} C_VEL
LIN {X 0,Y 347.927,Z 1144.795,A -85,B 0,C 180,E1 17289.929,E2 17289.929} C_VEL
LIN {X 0,Y 350.309,Z 1140.109,A -85,B 0,C 180,E1 17285.569,E2 17285.569} C_VEL
LIN {X 0,Y 353.758,Z 1133.786,A -85,B 0,C 180,E1 17281.296,E2 17281.296} C_VEL
LIN {X 0,Y 357.46,Z 1127.684,A -85,B 0,C 180,E1 17277.916,E2 17277.916} C_VEL
LIN {X 0,Y 363.212,Z 1118.815,A -85,B 0,C 180,E1 17273.837,E2 17273.837} C_VEL
LIN {X 0,Y 370.215,Z 1108.099,A -85,B 0,C 180,E1 17269.889,E2 17269.889} C_VEL
LIN {X 0,Y 377.549,Z 1097.249,A -85,B 0,C 180,E1 17266.523,E2 17266.523} C_VEL
LIN {X 0,Y 387.301,Z 1082.757,A -85,B 0,C 180,E1 17262.787,E2 17262.787} C_VEL
LIN {X 0,Y 396.555,Z 1068.981,A -85,B 0,C 180,E1 17259.791,E2 17259.791} C_VEL
LIN {X 0,Y 408.537,Z 1050.912,A -85,B 0,C 180,E1 17256.488,E2 17256.488} C_VEL
LIN {X 0,Y 420.931,Z 1032.418,A -85,B 0,C 180,E1 17253.627,E2 17253.627} C_VEL
LIN {X 0,Y 436.703,Z 1009.691,A -85,B 0,C 180,E1 17250.66,E2 17250.66} C_VEL
LIN {X 0,Y 440.749,Z 1004.032,A -85,B 0,C 180,E1 17249.995,E2 17249.995} C_VEL
LIN {X 0,Y 425.719,Z 1030.194,A -85,B 0,C 180,E1 17247.854,E2 17247.854} C_VEL
LIN {X 0,Y 409.78,Z 1063.795,A -85,B 0,C 180,E1 17244.705,E2 17244.705} C_VEL
LIN {X 0,Y 396.556,Z 1095.079,A -85,B 0,C 180,E1 17241.294,E2 17241.294} C_VEL
LIN {X 0,Y 386.277,Z 1121.317,A -85,B 0,C 180,E1 17237.979,E2 17237.979} C_VEL
LIN {X 0,Y 378.197,Z 1142.391,A -85,B 0,C 180,E1 17234.883,E2 17234.883} C_VEL
LIN {X 0,Y 372.169,Z 1158.549,A -85,B 0,C 180,E1 17232.195,E2 17232.195} C_VEL
LIN {X 0,Y 366.815,Z 1173.335,A -85,B 0,C 180,E1 17229.429,E2 17229.429} C_VEL
LIN {X 0,Y 362.14,Z 1186.744,A -85,B 0,C 180,E1 17226.611,E2 17226.611} C_VEL
LIN {X 0,Y 357.944,Z 1199.543,A -85,B 0,C 180,E1 17223.579,E2 17223.579} C_VEL
LIN {X 0,Y 354.396,Z 1210.963,A -85,B 0,C 180,E1 17220.52,E2 17220.52} C_VEL
LIN {X 0,Y 351.537,Z 1221.101,A -85,B 0,C 180,E1 17217.437,E2 17217.437} C_VEL
LIN {X 0,Y 349.209,Z 1230.569,A -85,B 0,C 180,E1 17214.17,E2 17214.17} C_VEL
LIN {X 0,Y 347.282,Z 1239.903,A -85,B 0,C 180,E1 17210.388,E2 17210.388} C_VEL
LIN {X 0,Y 346.005,Z 1248.59,A -85,B 0,C 180,E1 17206.106,E2 17206.106} C_VEL
LIN {X 0,Y 345.466,Z 1254.739,A -85,B 0,C 180,E1 17202.197,E2 17202.197} C_VEL
LIN {X 0,Y 345.291,Z 1258.633,A -85,B 0,C 180,E1 17198.996,E2 17198.996} C_VEL
LIN {X 0,Y 345.347,Z 1261.471,A -85,B 0,C 180,E1 17195.816,E2 17195.816} C_VEL
LIN {X 0,Y 345.392,Z 1263.274,A -85,B 0,C 180,E1 17192.489,E2 17192.489} C_VEL
LIN {X 0,Y 345.321,Z 1263.884,A -85,B 0,C 180,E1 17189.336,E2 17189.336} C_VEL
LIN {X 0,Y 345.255,Z 1263.435,A -85,B 0,C 180,E1 17186.181,E2 17186.181} C_VEL
LIN {X 0,Y 345.114,Z 1261.806,A -85,B 0,C 180,E1 17182.843,E2 17182.843} C_VEL
LIN {X 0,Y 345.099,Z 1258.851,A -85,B 0,C 180,E1 17179.314,E2 17179.314} C_VEL
LIN {X 0,Y 345.309,Z 1255.091,A -85,B 0,C 180,E1 17176.094,E2 17176.094} C_VEL
LIN {X 0,Y 345.939,Z 1250.288,A -85,B 0,C 180,E1 17172.854,E2 17172.854} C_VEL
LIN {X 0,Y 347.078,Z 1244.065,A -85,B 0,C 180,E1 17169.423,E2 17169.423} C_VEL
LIN {X 0,Y 348.796,Z 1237.046,A -85,B 0,C 180,E1 17166.159,E2 17166.159} C_VEL
LIN {X 0,Y 351.194,Z 1228.902,A -85,B 0,C 180,E1 17162.901,E2 17162.901} C_VEL
LIN {X 0,Y 354.687,Z 1218.472,A -85,B 0,C 180,E1 17159.297,E2 17159.297} C_VEL
LIN {X 0,Y 360.302,Z 1203.497,A -85,B 0,C 180,E1 17154.952,E2 17154.952} C_VEL
LIN {X 0,Y 365.578,Z 1190.38,A -85,B 0,C 180,E1 17151.718,E2 17151.718} C_VEL
LIN {X 0,Y 371.078,Z 1177.314,A -85,B 0,C 180,E1 17148.893,E2 17148.893} C_VEL
LIN {X 0,Y 378.815,Z 1159.431,A -85,B 0,C 180,E1 17145.522,E2 17145.522} C_VEL
LIN {X 0,Y 386.784,Z 1140.637,A -85,B 0,C 180,E1 17142.544,E2 17142.544} C_VEL
LIN {X 0,Y 393.771,Z 1124.136,A -85,B 0,C 180,E1 17140.267,E2 17140.267} C_VEL
LIN {X 0,Y 401.309,Z 1105.925,A -85,B 0,C 180,E1 17138.064,E2 17138.064} C_VEL
LIN {X 0,Y 410.928,Z 1081.652,A -85,B 0,C 180,E1 17135.56,E2 17135.56} C_VEL
LIN {X 0,Y 418.59,Z 1061.205,A -85,B 0,C 180,E1 17133.772,E2 17133.772} C_VEL
LIN {X 0,Y 425.428,Z 1041.932,A -85,B 0,C 180,E1 17132.312,E2 17132.312} C_VEL
LIN {X 0,Y 433.368,Z 1017.942,A -85,B 0,C 180,E1 17130.746,E2 17130.746} C_VEL
LIN {X 0,Y 441.074,Z 991.885,A -85,B 0,C 180,E1 17129.352,E2 17129.352} C_VEL
LIN {X 0,Y 446.749,Z 970.848,A -85,B 0,C 180,E1 17128.408,E2 17128.408} C_VEL
LIN {X 0,Y 452.258,Z 948.184,A -85,B 0,C 180,E1 17127.557,E2 17127.557} C_VEL
LIN {X 0,Y 458.444,Z 918.338,A -85,B 0,C 180,E1 17126.67,E2 17126.67} C_VEL
LIN {X 0,Y 462.264,Z 894.682,A -85,B 0,C 180,E1 17126.106,E2 17126.106} C_VEL
LIN {X 0,Y 464.967,Z 871.924,A -85,B 0,C 180,E1 17125.641,E2 17125.641} C_VEL
LIN {X 0,Y 485.271,Z 646.95,A -85,B 0,C 180,E1 17121.729,E2 17121.729} C_VEL
LIN {X 0,Y 493.046,Z 565.532,A -85,B 0,C 180,E1 17120.322,E2 17120.322} C_VEL
LIN {X 0,Y 483.182,Z 549.158,A -85,B 0,C 180,E1 17117.368,E2 17117.368} C_VEL
LIN {X 0,Y 473.59,Z 533.95,A -85,B 0,C 180,E1 17114.177,E2 17114.177} C_VEL
LIN {X 0,Y 464.666,Z 520.435,A -85,B 0,C 180,E1 17110.853,E2 17110.853} C_VEL
LIN {X 0,Y 456.086,Z 507.685,A -85,B 0,C 180,E1 17107.242,E2 17107.242} C_VEL
LIN {X 0,Y 448.716,Z 497.166,A -85,B 0,C 180,E1 17103.705,E2 17103.705} C_VEL
LIN {X 0,Y 443.808,Z 490.269,A -85,B 0,C 180,E1 17101.033,E2 17101.033} C_VEL
LIN {X 0,Y 440.395,Z 485.539,A -85,B 0,C 180,E1 17099.024,E2 17099.024} C_VEL
LIN {X 0,Y 436.941,Z 480.643,A -85,B 0,C 180,E1 17096.786,E2 17096.786} C_VEL
LIN {X 0,Y 433.537,Z 475.773,A -85,B 0,C 180,E1 17094.308,E2 17094.308} C_VEL
LIN {X 0,Y 430.194,Z 470.948,A -85,B 0,C 180,E1 17091.58,E2 17091.58} C_VEL
LIN {X 0,Y 426.523,Z 465.802,A -85,B 0,C 180,E1 17088.163,E2 17088.163} C_VEL
LIN {X 0,Y 425.479,Z 464.349,A -85,B 0,C 180,E1 17087.1,E2 17087.1} C_VEL
LIN {X 0,Y 422.956,Z 460.828,A -85,B 0,C 180,E1 17084.187,E2 17084.187} C_VEL
LIN {X 0,Y 422.243,Z 459.718,A -85,B 0,C 180,E1 17083.208,E2 17083.208} C_VEL
LIN {X 0,Y 419.221,Z 457.319,A -85,B 0,C 180,E1 17079.037,E2 17079.037} C_VEL
LIN {X 0,Y 417.477,Z 454.181,A -85,B 0,C 180,E1 17075.371,E2 17075.371} C_VEL
LIN {X 0,Y 416.355,Z 453.149,A -85,B 0,C 180,E1 17072.542,E2 17072.542} C_VEL
LIN {X 0,Y 415.184,Z 452.551,A -85,B 0,C 180,E1 17068.169,E2 17068.169} C_VEL
LIN {X 0,Y 414.851,Z 452.307,A -85,B 0,C 180,E1 17063.292,E2 17063.292} C_VEL
LIN {X 0,Y 415.356,Z 452.615,A -85,B 0,C 180,E1 17059.278,E2 17059.278} C_VEL
LIN {X 0,Y 417.016,Z 453.419,A -85,B 0,C 180,E1 17054.396,E2 17054.396} C_VEL
LIN {X 0,Y 417.835,Z 454.574,A -85,B 0,C 180,E1 17052.519,E2 17052.519} C_VEL
LIN {X 0,Y 419.853,Z 457.828,A -85,B 0,C 180,E1 17048.853,E2 17048.853} C_VEL
LIN {X 0,Y 423.153,Z 460.281,A -85,B 0,C 180,E1 17044.795,E2 17044.795} C_VEL
LIN {X 0,Y 425.693,Z 464.27,A -85,B 0,C 180,E1 17042.012,E2 17042.012} C_VEL
LIN {X 0,Y 428.677,Z 466.733,A -85,B 0,C 180,E1 17039.482,E2 17039.482} C_VEL
LIN {X 0,Y 431.491,Z 470.791,A -85,B 0,C 180,E1 17037.146,E2 17037.146} C_VEL
LIN {X 0,Y 433.881,Z 472.989,A -85,B 0,C 180,E1 17035.527,E2 17035.527} C_VEL
LIN {X 0,Y 437.384,Z 477.429,A -85,B 0,C 180,E1 17033.219,E2 17033.219} C_VEL
LIN {X 0,Y 439.107,Z 479.168,A -85,B 0,C 180,E1 17032.209,E2 17032.209} C_VEL
LIN {X 0,Y 443.051,Z 483.946,A -85,B 0,C 180,E1 17029.993,E2 17029.993} C_VEL
LIN {X 0,Y 449.091,Z 491.384,A -85,B 0,C 180,E1 17026.958,E2 17026.958} C_VEL
LIN {X 0,Y 453.871,Z 497.352,A -85,B 0,C 180,E1 17024.806,E2 17024.806} C_VEL
LIN {X 0,Y 458.636,Z 503.428,A -85,B 0,C 180,E1 17022.816,E2 17022.816} C_VEL
LIN {X 0,Y 465.63,Z 512.325,A -85,B 0,C 180,E1 17020.173,E2 17020.173} C_VEL
LIN {X 0,Y 473.982,Z 523.506,A -85,B 0,C 180,E1 17017.313,E2 17017.313} C_VEL
LIN {X 0,Y 483.905,Z 537.118,A -85,B 0,C 180,E1 17014.266,E2 17014.266} C_VEL
LIN {X 0,Y 488.721,Z 544.4,A -85,B 0,C 180,E1 17012.875,E2 17012.875} C_VEL
LIN {X 0,Y 470.235,Z 747.419,A -85,B 0,C 180,E1 17009.418,E2 17009.418} C_VEL
LIN {X 0,Y 465.907,Z 792.414,A -85,B 0,C 180,E1 17008.596,E2 17008.596} C_VEL
LIN {X 0,Y 462.272,Z 818.592,A -85,B 0,C 180,E1 17007.938,E2 17007.938} C_VEL
LIN {X 0,Y 458.281,Z 841.947,A -85,B 0,C 180,E1 17007.203,E2 17007.203} C_VEL
LIN {X 0,Y 452.663,Z 869.306,A -85,B 0,C 180,E1 17006.143,E2 17006.143} C_VEL
LIN {X 0,Y 446.71,Z 893.531,A -85,B 0,C 180,E1 17004.992,E2 17004.992} C_VEL
LIN {X 0,Y 441.071,Z 914.056,A -85,B 0,C 180,E1 17003.848,E2 17003.848} C_VEL
LIN {X 0,Y 434.68,Z 935.02,A -85,B 0,C 180,E1 17002.494,E2 17002.494} C_VEL
LIN {X 0,Y 426.275,Z 959.698,A -85,B 0,C 180,E1 17000.618,E2 17000.618} C_VEL
LIN {X 0,Y 419.201,Z 978.675,A -85,B 0,C 180,E1 16998.93,E2 16998.93} C_VEL
LIN {X 0,Y 412.637,Z 995.185,A -85,B 0,C 180,E1 16997.261,E2 16997.261} C_VEL
LIN {X 0,Y 405.753,Z 1011.617,A -85,B 0,C 180,E1 16995.377,E2 16995.377} C_VEL
LIN {X 0,Y 397.199,Z 1031.172,A -85,B 0,C 180,E1 16992.795,E2 16992.795} C_VEL
LIN {X 0,Y 389.174,Z 1048.309,A -85,B 0,C 180,E1 16990.111,E2 16990.111} C_VEL
LIN {X 0,Y 382.641,Z 1061.851,A -85,B 0,C 180,E1 16987.676,E2 16987.676} C_VEL
LIN {X 0,Y 376.541,Z 1074.326,A -85,B 0,C 180,E1 16985.118,E2 16985.118} C_VEL
LIN {X 0,Y 375.265,Z 1077.011,A -85,B 0,C 180,E1 16984.53,E2 16984.53} C_VEL
LIN {X 0,Y 372.373,Z 1081.382,A -85,B 0,C 180,E1 16983.65,E2 16983.65} C_VEL
LIN {X 0,Y 362.084,Z 1092.376,A -85,B 0,C 180,E1 16981.557,E2 16981.557} C_VEL
LIN {X 0,Y 359.329,Z 1096.22,A -85,B 0,C 180,E1 16980.584,E2 16980.584} C_VEL
LIN {X 0,Y 354.029,Z 1106.87,A -85,B 0,C 180,E1 16977.315,E2 16977.315} C_VEL
LIN {X 0,Y 348.313,Z 1118.79,A -85,B 0,C 180,E1 16972.927,E2 16972.927} C_VEL
LIN {X 0,Y 344.801,Z 1126.611,A -85,B 0,C 180,E1 16969.445,E2 16969.445} C_VEL
LIN {X 0,Y 342.093,Z 1133.267,A -85,B 0,C 180,E1 16965.923,E2 16965.923} C_VEL
LIN {X 0,Y 340.109,Z 1138.906,A -85,B 0,C 180,E1 16962.318,E2 16962.318} C_VEL
LIN {X 0,Y 338.622,Z 1144.199,A -85,B 0,C 180,E1 16958.108,E2 16958.108} C_VEL
LIN {X 0,Y 337.805,Z 1148.036,A -85,B 0,C 180,E1 16953.813,E2 16953.813} C_VEL
LIN {X 0,Y 337.561,Z 1150.257,A -85,B 0,C 180,E1 16950.236,E2 16950.236} C_VEL
LIN {X 0,Y 337.456,Z 1151.568,A -85,B 0,C 180,E1 16946.893,E2 16946.893} C_VEL
LIN {X 0,Y 337.553,Z 1152.116,A -85,B 0,C 180,E1 16943.572,E2 16943.572} C_VEL
LIN {X 0,Y 337.763,Z 1151.922,A -85,B 0,C 180,E1 16940.214,E2 16940.214} C_VEL
LIN {X 0,Y 338.169,Z 1150.973,A -85,B 0,C 180,E1 16936.844,E2 16936.844} C_VEL
LIN {X 0,Y 338.864,Z 1149.276,A -85,B 0,C 180,E1 16933.48,E2 16933.48} C_VEL
LIN {X 0,Y 340.147,Z 1146.542,A -85,B 0,C 180,E1 16929.817,E2 16929.817} C_VEL
LIN {X 0,Y 342.148,Z 1142.741,A -85,B 0,C 180,E1 16926.039,E2 16926.039} C_VEL
LIN {X 0,Y 346.1,Z 1136.141,A -85,B 0,C 180,E1 16921.159,E2 16921.159} C_VEL
LIN {X 0,Y 350.325,Z 1129.58,A -85,B 0,C 180,E1 16917.383,E2 16917.383} C_VEL
LIN {X 0,Y 355.322,Z 1122.224,A -85,B 0,C 180,E1 16913.861,E2 16913.861} C_VEL
LIN {X 0,Y 363.409,Z 1110.732,A -85,B 0,C 180,E1 16909.377,E2 16909.377} C_VEL
LIN {X 0,Y 371.051,Z 1100.055,A -85,B 0,C 180,E1 16905.952,E2 16905.952} C_VEL
LIN {X 0,Y 381.316,Z 1085.757,A -85,B 0,C 180,E1 16902.134,E2 16902.134} C_VEL
LIN {X 0,Y 391.222,Z 1071.907,A -85,B 0,C 180,E1 16899.034,E2 16899.034} C_VEL
LIN {X 0,Y 404.256,Z 1053.641,A -85,B 0,C 180,E1 16895.603,E2 16895.603} C_VEL
LIN {X 0,Y 418.449,Z 1034.199,A -85,B 0,C 180,E1 16892.537,E2 16892.537} C_VEL
LIN {X 0,Y 432.008,Z 1016.545,A -85,B 0,C 180,E1 16890.157,E2 16890.157} C_VEL
LIN {X 0,Y 418.368,Z 1038.883,A -85,B 0,C 180,E1 16888.171,E2 16888.171} C_VEL
LIN {X 0,Y 402.768,Z 1069.035,A -85,B 0,C 180,E1 16885.132,E2 16885.132} C_VEL
LIN {X 0,Y 388.592,Z 1100.72,A -85,B 0,C 180,E1 16881.487,E2 16881.487} C_VEL
LIN {X 0,Y 378.76,Z 1124.149,A -85,B 0,C 180,E1 16878.338,E2 16878.338} C_VEL
LIN {X 0,Y 371.718,Z 1141.641,A -85,B 0,C 180,E1 16875.685,E2 16875.685} C_VEL
LIN {X 0,Y 365.413,Z 1157.705,A -85,B 0,C 180,E1 16872.948,E2 16872.948} C_VEL
LIN {X 0,Y 359.516,Z 1173.194,A -85,B 0,C 180,E1 16869.975,E2 16869.975} C_VEL
LIN {X 0,Y 353.661,Z 1189.456,A -85,B 0,C 180,E1 16866.421,E2 16866.421} C_VEL
LIN {X 0,Y 348.171,Z 1205.579,A -85,B 0,C 180,E1 16862.286,E2 16862.286} C_VEL
LIN {X 0,Y 344.617,Z 1217.275,A -85,B 0,C 180,E1 16858.792,E2 16858.792} C_VEL
LIN {X 0,Y 342.119,Z 1226.531,A -85,B 0,C 180,E1 16855.629,E2 16855.629} C_VEL
LIN {X 0,Y 340.079,Z 1235.499,A -85,B 0,C 180,E1 16852.107,E2 16852.107} C_VEL
LIN {X 0,Y 338.662,Z 1243.089,A -85,B 0,C 180,E1 16848.594,E2 16848.594} C_VEL
LIN {X 0,Y 337.89,Z 1249.115,A -85,B 0,C 180,E1 16845.267,E2 16845.267} C_VEL
LIN {X 0,Y 337.51,Z 1254.224,A -85,B 0,C 180,E1 16841.795,E2 16841.795} C_VEL
LIN {X 0,Y 337.388,Z 1257.922,A -85,B 0,C 180,E1 16838.521,E2 16838.521} C_VEL
LIN {X 0,Y 337.453,Z 1260.322,A -85,B 0,C 180,E1 16835.611,E2 16835.611} C_VEL
LIN {X 0,Y 337.5,Z 1261.927,A -85,B 0,C 180,E1 16832.547,E2 16832.547} C_VEL
LIN {X 0,Y 337.432,Z 1262.556,A -85,B 0,C 180,E1 16829.321,E2 16829.321} C_VEL
LIN {X 0,Y 337.355,Z 1262.118,A -85,B 0,C 180,E1 16826.091,E2 16826.091} C_VEL
LIN {X 0,Y 337.192,Z 1260.482,A -85,B 0,C 180,E1 16822.674,E2 16822.674} C_VEL
LIN {X 0,Y 337.172,Z 1257.684,A -85,B 0,C 180,E1 16819.232,E2 16819.232} C_VEL
LIN {X 0,Y 337.378,Z 1253.955,A -85,B 0,C 180,E1 16815.935,E2 16815.935} C_VEL
LIN {X 0,Y 338.03,Z 1249.181,A -85,B 0,C 180,E1 16812.617,E2 16812.617} C_VEL
LIN {X 0,Y 339.218,Z 1242.988,A -85,B 0,C 180,E1 16809.105,E2 16809.105} C_VEL
LIN {X 0,Y 341.012,Z 1235.994,A -85,B 0,C 180,E1 16805.764,E2 16805.764} C_VEL
LIN {X 0,Y 343.517,Z 1227.855,A -85,B 0,C 180,E1 16802.432,E2 16802.432} C_VEL
LIN {X 0,Y 347.145,Z 1217.467,A -85,B 0,C 180,E1 16798.772,E2 16798.772} C_VEL
LIN {X 0,Y 352.877,Z 1202.788,A -85,B 0,C 180,E1 16794.413,E2 16794.413} C_VEL
LIN {X 0,Y 358.367,Z 1189.69,A -85,B 0,C 180,E1 16791.114,E2 16791.114} C_VEL
LIN {X 0,Y 363.885,Z 1177.032,A -85,B 0,C 180,E1 16788.32,E2 16788.32} C_VEL
LIN {X 0,Y 370.885,Z 1161.266,A -85,B 0,C 180,E1 16785.281,E2 16785.281} C_VEL
LIN {X 0,Y 379.781,Z 1141.115,A -85,B 0,C 180,E1 16781.97,E2 16781.97} C_VEL
LIN {X 0,Y 387.221,Z 1124.09,A -85,B 0,C 180,E1 16779.576,E2 16779.576} C_VEL
LIN {X 0,Y 394.562,Z 1106.907,A -85,B 0,C 180,E1 16777.46,E2 16777.46} C_VEL
LIN {X 0,Y 402.973,Z 1086.545,A -85,B 0,C 180,E1 16775.281,E2 16775.281} C_VEL
LIN {X 0,Y 412.061,Z 1063.024,A -85,B 0,C 180,E1 16773.16,E2 16773.16} C_VEL
LIN {X 0,Y 419.571,Z 1042.422,A -85,B 0,C 180,E1 16771.575,E2 16771.575} C_VEL
LIN {X 0,Y 426.764,Z 1021.282,A -85,B 0,C 180,E1 16770.17,E2 16770.17} C_VEL
LIN {X 0,Y 435.5,Z 993.078,A -85,B 0,C 180,E1 16768.613,E2 16768.613} C_VEL
LIN {X 0,Y 441.544,Z 971.318,A -85,B 0,C 180,E1 16767.627,E2 16767.627} C_VEL
LIN {X 0,Y 446.971,Z 949.637,A -85,B 0,C 180,E1 16766.803,E2 16766.803} C_VEL
LIN {X 0,Y 452.945,Z 922.484,A -85,B 0,C 180,E1 16765.964,E2 16765.964} C_VEL
LIN {X 0,Y 457.584,Z 894.985,A -85,B 0,C 180,E1 16765.298,E2 16765.298} C_VEL
LIN {X 0,Y 460.446,Z 871.781,A -85,B 0,C 180,E1 16764.82,E2 16764.82} C_VEL
LIN {X 0,Y 481.698,Z 643.38,A -85,B 0,C 180,E1 16760.837,E2 16760.837} C_VEL
LIN {X 0,Y 488.847,Z 569.99,A -85,B 0,C 180,E1 16759.569,E2 16759.569} C_VEL
LIN {X 0,Y 479.331,Z 554.207,A -85,B 0,C 180,E1 16756.637,E2 16756.637} C_VEL
LIN {X 0,Y 470.297,Z 539.804,A -85,B 0,C 180,E1 16753.556,E2 16753.556} C_VEL
LIN {X 0,Y 461.685,Z 526.73,A -85,B 0,C 180,E1 16750.293,E2 16750.293} C_VEL
LIN {X 0,Y 453.932,Z 515.057,A -85,B 0,C 180,E1 16746.958,E2 16746.958} C_VEL
LIN {X 0,Y 446.766,Z 504.715,A -85,B 0,C 180,E1 16743.476,E2 16743.476} C_VEL
LIN {X 0,Y 441.853,Z 497.773,A -85,B 0,C 180,E1 16740.778,E2 16740.778} C_VEL
LIN {X 0,Y 438.509,Z 493.051,A -85,B 0,C 180,E1 16738.759,E2 16738.759} C_VEL
LIN {X 0,Y 435.152,Z 488.275,A -85,B 0,C 180,E1 16736.575,E2 16736.575} C_VEL
LIN {X 0,Y 431.64,Z 483.305,A -85,B 0,C 180,E1 16734.016,E2 16734.016} C_VEL
LIN {X 0,Y 427.647,Z 477.672,A -85,B 0,C 180,E1 16730.716,E2 16730.716} C_VEL
LIN {X 0,Y 424.761,Z 473.372,A -85,B 0,C 180,E1 16727.906,E2 16727.906} C_VEL
LIN {X 0,Y 423.043,Z 471.185,A -85,B 0,C 180,E1 16726.049,E2 16726.049} C_VEL
LIN {X 0,Y 420.708,Z 467.557,A -85,B 0,C 180,E1 16723.145,E2 16723.145} C_VEL
LIN {X 0,Y 417.653,Z 465.141,A -85,B 0,C 180,E1 16718.954,E2 16718.954} C_VEL
LIN {X 0,Y 415.972,Z 462.16,A -85,B 0,C 180,E1 16715.427,E2 16715.427} C_VEL
LIN {X 0,Y 415.076,Z 461.088,A -85,B 0,C 180,E1 16713.071,E2 16713.071} C_VEL
LIN {X 0,Y 413.74,Z 460.481,A -85,B 0,C 180,E1 16708.695,E2 16708.695} C_VEL
LIN {X 0,Y 413.385,Z 460.169,A -85,B 0,C 180,E1 16704.343,E2 16704.343} C_VEL
LIN {X 0,Y 413.701,Z 460.392,A -85,B 0,C 180,E1 16699.991,E2 16699.991} C_VEL
LIN {X 0,Y 414.981,Z 461.012,A -85,B 0,C 180,E1 16695.673,E2 16695.673} C_VEL
LIN {X 0,Y 416.079,Z 461.951,A -85,B 0,C 180,E1 16693.067,E2 16693.067} C_VEL
LIN {X 0,Y 417.61,Z 464.863,A -85,B 0,C 180,E1 16689.916,E2 16689.916} C_VEL
LIN {X 0,Y 420.931,Z 467.539,A -85,B 0,C 180,E1 16685.669,E2 16685.669} C_VEL
LIN {X 0,Y 421.615,Z 468.222,A -85,B 0,C 180,E1 16684.858,E2 16684.858} C_VEL
LIN {X 0,Y 424.279,Z 472.244,A -85,B 0,C 180,E1 16681.961,E2 16681.961} C_VEL
LIN {X 0,Y 426.961,Z 474.428,A -85,B 0,C 180,E1 16679.676,E2 16679.676} C_VEL
LIN {X 0,Y 429.866,Z 478.568,A -85,B 0,C 180,E1 16677.273,E2 16677.273} C_VEL
LIN {X 0,Y 432.156,Z 480.708,A -85,B 0,C 180,E1 16675.71,E2 16675.71} C_VEL
LIN {X 0,Y 435.689,Z 485.167,A -85,B 0,C 180,E1 16673.366,E2 16673.366} C_VEL
LIN {X 0,Y 437.371,Z 486.931,A -85,B 0,C 180,E1 16672.373,E2 16672.373} C_VEL
LIN {X 0,Y 441.473,Z 491.803,A -85,B 0,C 180,E1 16670.067,E2 16670.067} C_VEL
LIN {X 0,Y 447.278,Z 499.116,A -85,B 0,C 180,E1 16667.129,E2 16667.129} C_VEL
LIN {X 0,Y 451.865,Z 504.887,A -85,B 0,C 180,E1 16665.041,E2 16665.041} C_VEL
LIN {X 0,Y 456.99,Z 511.447,A -85,B 0,C 180,E1 16662.895,E2 16662.895} C_VEL
LIN {X 0,Y 464.162,Z 520.747,A -85,B 0,C 180,E1 16660.174,E2 16660.174} C_VEL
LIN {X 0,Y 472.276,Z 531.656,A -85,B 0,C 180,E1 16657.39,E2 16657.39} C_VEL
LIN {X 0,Y 481.713,Z 544.785,A -85,B 0,C 180,E1 16654.464,E2 16654.464} C_VEL
LIN {X 0,Y 484.568,Z 549.315,A -85,B 0,C 180,E1 16653.632,E2 16653.632} C_VEL
LIN {X 0,Y 465.281,Z 754.869,A -85,B 0,C 180,E1 16650.119,E2 16650.119} C_VEL
LIN {X 0,Y 461.261,Z 794.644,A -85,B 0,C 180,E1 16649.379,E2 16649.379} C_VEL
LIN {X 0,Y 457.631,Z 820.026,A -85,B 0,C 180,E1 16648.735,E2 16648.735} C_VEL
LIN {X 0,Y 453.489,Z 843.624,A -85,B 0,C 180,E1 16647.986,E2 16647.986} C_VEL
LIN {X 0,Y 447.428,Z 872.085,A -85,B 0,C 180,E1 16646.868,E2 16646.868} C_VEL
LIN {X 0,Y 441.708,Z 894.788,A -85,B 0,C 180,E1 16645.781,E2 16645.781} C_VEL
LIN {X 0,Y 435.782,Z 915.822,A -85,B 0,C 180,E1 16644.602,E2 16644.602} C_VEL
LIN {X 0,Y 428.26,Z 939.924,A -85,B 0,C 180,E1 16643.027,E2 16643.027} C_VEL
LIN {X 0,Y 420.156,Z 962.809,A -85,B 0,C 180,E1 16641.24,E2 16641.24} C_VEL
LIN {X 0,Y 413.593,Z 980.003,A -85,B 0,C 180,E1 16639.695,E2 16639.695} C_VEL
LIN {X 0,Y 406.554,Z 997.255,A -85,B 0,C 180,E1 16637.933,E2 16637.933} C_VEL
LIN {X 0,Y 398.321,Z 1016.401,A -85,B 0,C 180,E1 16635.689,E2 16635.689} C_VEL
LIN {X 0,Y 389.29,Z 1035.992,A -85,B 0,C 180,E1 16632.974,E2 16632.974} C_VEL
LIN {X 0,Y 382.178,Z 1050.806,A -85,B 0,C 180,E1 16630.594,E2 16630.594} C_VEL
LIN {X 0,Y 375.48,Z 1064.355,A -85,B 0,C 180,E1 16628.111,E2 16628.111} C_VEL
LIN {X 0,Y 368.749,Z 1077.776,A -85,B 0,C 180,E1 16625.283,E2 16625.283} C_VEL
LIN {X 0,Y 360.874,Z 1093.184,A -85,B 0,C 180,E1 16621.442,E2 16621.442} C_VEL
LIN {X 0,Y 359.329,Z 1096.22,A -85,B 0,C 180,E1 16620.584,E2 16620.584} C_VEL
LIN {X 0,Y 356.641,Z 1100.123,A -85,B 0,C 180,E1 16619.592,E2 16619.592} C_VEL
LIN {X 0,Y 346.369,Z 1110.296,A -85,B 0,C 180,E1 16617.051,E2 16617.051} C_VEL
LIN {X 0,Y 344.292,Z 1113.061,A -85,B 0,C 180,E1 16616.113,E2 16616.113} C_VEL
LIN {X 0,Y 340.202,Z 1121.417,A -85,B 0,C 180,E1 16612.797,E2 16612.797} C_VEL
LIN {X 0,Y 336.879,Z 1128.642,A -85,B 0,C 180,E1 16609.45,E2 16609.45} C_VEL
LIN {X 0,Y 334.275,Z 1134.857,A -85,B 0,C 180,E1 16606.056,E2 16606.056} C_VEL
LIN {X 0,Y 332.252,Z 1140.448,A -85,B 0,C 180,E1 16602.386,E2 16602.386} C_VEL
LIN {X 0,Y 330.665,Z 1145.897,A -85,B 0,C 180,E1 16597.869,E2 16597.869} C_VEL
LIN {X 0,Y 329.92,Z 1149.361,A -85,B 0,C 180,E1 16593.86,E2 16593.86} C_VEL
LIN {X 0,Y 329.667,Z 1151.599,A -85,B 0,C 180,E1 16590.186,E2 16590.186} C_VEL
LIN {X 0,Y 329.575,Z 1152.929,A -85,B 0,C 180,E1 16586.681,E2 16586.681} C_VEL
LIN {X 0,Y 329.663,Z 1153.463,A -85,B 0,C 180,E1 16583.412,E2 16583.412} C_VEL
LIN {X 0,Y 329.905,Z 1153.294,A -85,B 0,C 180,E1 16580.025,E2 16580.025} C_VEL
LIN {X 0,Y 330.355,Z 1152.374,A -85,B 0,C 180,E1 16576.53,E2 16576.53} C_VEL
LIN {X 0,Y 331.115,Z 1150.71,A -85,B 0,C 180,E1 16573.09,E2 16573.09} C_VEL
LIN {X 0,Y 332.487,Z 1148.108,A -85,B 0,C 180,E1 16569.468,E2 16569.468} C_VEL
LIN {X 0,Y 334.588,Z 1144.429,A -85,B 0,C 180,E1 16565.659,E2 16565.659} C_VEL
LIN {X 0,Y 338.443,Z 1138.499,A -85,B 0,C 180,E1 16561.016,E2 16561.016} C_VEL
LIN {X 0,Y 343.017,Z 1131.822,A -85,B 0,C 180,E1 16556.992,E2 16556.992} C_VEL
LIN {X 0,Y 348.491,Z 1124.285,A -85,B 0,C 180,E1 16553.244,E2 16553.244} C_VEL
LIN {X 0,Y 356.97,Z 1112.977,A -85,B 0,C 180,E1 16548.693,E2 16548.693} C_VEL
LIN {X 0,Y 364.555,Z 1102.989,A -85,B 0,C 180,E1 16545.384,E2 16545.384} C_VEL
LIN {X 0,Y 374.447,Z 1090.235,A -85,B 0,C 180,E1 16541.794,E2 16541.794} C_VEL
LIN {X 0,Y 386.019,Z 1074.971,A -85,B 0,C 180,E1 16538.259,E2 16538.259} C_VEL
LIN {X 0,Y 400.187,Z 1056.604,A -85,B 0,C 180,E1 16534.707,E2 16534.707} C_VEL
LIN {X 0,Y 416.366,Z 1036.412,A -85,B 0,C 180,E1 16531.452,E2 16531.452} C_VEL
LIN {X 0,Y 423.171,Z 1028.438,A -85,B 0,C 180,E1 16530.3,E2 16530.3} C_VEL
LIN {X 0,Y 410.004,Z 1048.732,A -85,B 0,C 180,E1 16528.332,E2 16528.332} C_VEL
LIN {X 0,Y 396.116,Z 1073.969,A -85,B 0,C 180,E1 16525.63,E2 16525.63} C_VEL
LIN {X 0,Y 381.272,Z 1104.575,A -85,B 0,C 180,E1 16521.882,E2 16521.882} C_VEL
LIN {X 0,Y 371.498,Z 1126.622,A -85,B 0,C 180,E1 16518.787,E2 16518.787} C_VEL
LIN {X 0,Y 361.303,Z 1150.636,A -85,B 0,C 180,E1 16514.885,E2 16514.885} C_VEL
LIN {X 0,Y 354.527,Z 1167.343,A -85,B 0,C 180,E1 16511.728,E2 16511.728} C_VEL
LIN {X 0,Y 348.943,Z 1181.704,A -85,B 0,C 180,E1 16508.658,E2 16508.658} C_VEL
LIN {X 0,Y 344.124,Z 1194.66,A -85,B 0,C 180,E1 16505.529,E2 16505.529} C_VEL
LIN {X 0,Y 340.28,Z 1205.752,A -85,B 0,C 180,E1 16502.506,E2 16502.506} C_VEL
LIN {X 0,Y 337.008,Z 1216.141,A -85,B 0,C 180,E1 16499.31,E2 16499.31} C_VEL
LIN {X 0,Y 334.385,Z 1225.389,A -85,B 0,C 180,E1 16496.076,E2 16496.076} C_VEL
LIN {X 0,Y 332.418,Z 1233.477,A -85,B 0,C 180,E1 16492.831,E2 16492.831} C_VEL
LIN {X 0,Y 330.967,Z 1240.859,A -85,B 0,C 180,E1 16489.409,E2 16489.409} C_VEL
LIN {X 0,Y 330.047,Z 1247.345,A -85,B 0,C 180,E1 16485.822,E2 16485.822} C_VEL
LIN {X 0,Y 329.604,Z 1252.558,A -85,B 0,C 180,E1 16482.26,E2 16482.26} C_VEL
LIN {X 0,Y 329.459,Z 1256.207,A -85,B 0,C 180,E1 16479.08,E2 16479.08} C_VEL
LIN {X 0,Y 329.548,Z 1258.981,A -85,B 0,C 180,E1 16475.746,E2 16475.746} C_VEL
LIN {X 0,Y 329.605,Z 1260.601,A -85,B 0,C 180,E1 16472.608,E2 16472.608} C_VEL
LIN {X 0,Y 329.541,Z 1261.234,A -85,B 0,C 180,E1 16469.305,E2 16469.305} C_VEL
LIN {X 0,Y 329.456,Z 1260.794,A -85,B 0,C 180,E1 16465.997,E2 16465.997} C_VEL
LIN {X 0,Y 329.28,Z 1259.27,A -85,B 0,C 180,E1 16462.673,E2 16462.673} C_VEL
LIN {X 0,Y 329.244,Z 1256.517,A -85,B 0,C 180,E1 16459.147,E2 16459.147} C_VEL
LIN {X 0,Y 329.469,Z 1252.593,A -85,B 0,C 180,E1 16455.59,E2 16455.59} C_VEL
LIN {X 0,Y 330.161,Z 1247.794,A -85,B 0,C 180,E1 16452.189,E2 16452.189} C_VEL
LIN {X 0,Y 331.455,Z 1241.56,A -85,B 0,C 180,E1 16448.592,E2 16448.592} C_VEL
LIN {X 0,Y 333.364,Z 1234.506,A -85,B 0,C 180,E1 16445.171,E2 16445.171} C_VEL
LIN {X 0,Y 336.159,Z 1225.844,A -85,B 0,C 180,E1 16441.582,E2 16441.582} C_VEL
LIN {X 0,Y 340.713,Z 1213.774,A -85,B 0,C 180,E1 16437.318,E2 16437.318} C_VEL
LIN {X 0,Y 346.346,Z 1200.035,A -85,B 0,C 180,E1 16433.302,E2 16433.302} C_VEL
LIN {X 0,Y 351.952,Z 1187.286,A -85,B 0,C 180,E1 16430.092,E2 16430.092} C_VEL
LIN {X 0,Y 358.531,Z 1172.749,A -85,B 0,C 180,E1 16426.901,E2 16426.901} C_VEL
LIN {X 0,Y 367.373,Z 1153.445,A -85,B 0,C 180,E1 16423.305,E2 16423.305} C_VEL
LIN {X 0,Y 374.748,Z 1137.303,A -85,B 0,C 180,E1 16420.734,E2 16420.734} C_VEL
LIN {X 0,Y 381.966,Z 1121.212,A -85,B 0,C 180,E1 16418.492,E2 16418.492} C_VEL
LIN {X 0,Y 391.045,Z 1100.486,A -85,B 0,C 180,E1 16415.988,E2 16415.988} C_VEL
LIN {X 0,Y 400.294,Z 1078.077,A -85,B 0,C 180,E1 16413.718,E2 16413.718} C_VEL
LIN {X 0,Y 407.978,Z 1058.468,A -85,B 0,C 180,E1 16412.007,E2 16412.007} C_VEL
LIN {X 0,Y 416.039,Z 1036.679,A -85,B 0,C 180,E1 16410.368,E2 16410.368} C_VEL
LIN {X 0,Y 425.134,Z 1009.786,A -85,B 0,C 180,E1 16408.686,E2 16408.686} C_VEL
LIN {X 0,Y 431.9,Z 987.765,A -85,B 0,C 180,E1 16407.542,E2 16407.542} C_VEL
LIN {X 0,Y 438.367,Z 964.579,A -85,B 0,C 180,E1 16406.532,E2 16406.532} C_VEL
LIN {X 0,Y 445.446,Z 935.236,A -85,B 0,C 180,E1 16405.512,E2 16405.512} C_VEL
LIN {X 0,Y 450.222,Z 911.71,A -85,B 0,C 180,E1 16404.87,E2 16404.87} C_VEL
LIN {X 0,Y 454.11,Z 887.281,A -85,B 0,C 180,E1 16404.3,E2 16404.3} C_VEL
LIN {X 0,Y 458.129,Z 849.643,A -85,B 0,C 180,E1 16403.587,E2 16403.587} C_VEL
LIN {X 0,Y 478.39,Z 637.493,A -85,B 0,C 180,E1 16399.898,E2 16399.898} C_VEL
LIN {X 0,Y 484.651,Z 574.481,A -85,B 0,C 180,E1 16398.806,E2 16398.806} C_VEL
LIN {X 0,Y 476.152,Z 560.375,A -85,B 0,C 180,E1 16396.124,E2 16396.124} C_VEL
LIN {X 0,Y 467.799,Z 546.892,A -85,B 0,C 180,E1 16393.221,E2 16393.221} C_VEL
LIN {X 0,Y 459.643,Z 534.36,A -85,B 0,C 180,E1 16390.085,E2 16390.085} C_VEL
LIN {X 0,Y 451.998,Z 522.742,A -85,B 0,C 180,E1 16386.768,E2 16386.768} C_VEL
LIN {X 0,Y 445.023,Z 512.51,A -85,B 0,C 180,E1 16383.349,E2 16383.349} C_VEL
LIN {X 0,Y 439.662,Z 504.967,A -85,B 0,C 180,E1 16380.391,E2 16380.391} C_VEL
LIN {X 0,Y 436.521,Z 500.423,A -85,B 0,C 180,E1 16378.425,E2 16378.425} C_VEL
LIN {X 0,Y 433.265,Z 495.783,A -85,B 0,C 180,E1 16376.295,E2 16376.295} C_VEL
LIN {X 0,Y 429.756,Z 490.83,A -85,B 0,C 180,E1 16373.722,E2 16373.722} C_VEL
LIN {X 0,Y 425.961,Z 485.389,A -85,B 0,C 180,E1 16370.542,E2 16370.542} C_VEL
LIN {X 0,Y 423.135,Z 481.205,A -85,B 0,C 180,E1 16367.79,E2 16367.79} C_VEL
LIN {X 0,Y 421.827,Z 479.434,A -85,B 0,C 180,E1 16366.371,E2 16366.371} C_VEL
LIN {X 0,Y 419.151,Z 475.383,A -85,B 0,C 180,E1 16363.053,E2 16363.053} C_VEL
LIN {X 0,Y 416.087,Z 472.964,A -85,B 0,C 180,E1 16358.871,E2 16358.871} C_VEL
LIN {X 0,Y 414.452,Z 470.09,A -85,B 0,C 180,E1 16355.439,E2 16355.439} C_VEL
LIN {X 0,Y 413.801,Z 469.078,A -85,B 0,C 180,E1 16353.601,E2 16353.601} C_VEL
LIN {X 0,Y 412.298,Z 468.363,A -85,B 0,C 180,E1 16349.06,E2 16349.06} C_VEL
LIN {X 0,Y 411.83,Z 468.044,A -85,B 0,C 180,E1 16345.147,E2 16345.147} C_VEL
LIN {X 0,Y 412.143,Z 468.218,A -85,B 0,C 180,E1 16340.269,E2 16340.269} C_VEL
LIN {X 0,Y 413.259,Z 468.804,A -85,B 0,C 180,E1 16336.138,E2 16336.138} C_VEL
LIN {X 0,Y 414.414,Z 469.554,A -85,B 0,C 180,E1 16333.427,E2 16333.427} C_VEL
LIN {X 0,Y 415.997,Z 472.603,A -85,B 0,C 180,E1 16330.102,E2 16330.102} C_VEL
LIN {X 0,Y 419.093,Z 475.244,A -85,B 0,C 180,E1 16326.021,E2 16326.021} C_VEL
LIN {X 0,Y 420.01,Z 475.999,A -85,B 0,C 180,E1 16325.01,E2 16325.01} C_VEL
LIN {X 0,Y 422.645,Z 479.994,A -85,B 0,C 180,E1 16322.118,E2 16322.118} C_VEL
LIN {X 0,Y 425.299,Z 482.214,A -85,B 0,C 180,E1 16319.827,E2 16319.827} C_VEL
LIN {X 0,Y 428.266,Z 486.367,A -85,B 0,C 180,E1 16317.383,E2 16317.383} C_VEL
LIN {X 0,Y 430.436,Z 488.426,A -85,B 0,C 180,E1 16315.894,E2 16315.894} C_VEL
LIN {X 0,Y 434.181,Z 493.065,A -85,B 0,C 180,E1 16313.406,E2 16313.406} C_VEL
LIN {X 0,Y 435.775,Z 494.9,A -85,B 0,C 180,E1 16312.452,E2 16312.452} C_VEL
LIN {X 0,Y 440.567,Z 500.791,A -85,B 0,C 180,E1 16309.765,E2 16309.765} C_VEL
LIN {X 0,Y 445.32,Z 506.638,A -85,B 0,C 180,E1 16307.375,E2 16307.375} C_VEL
LIN {X 0,Y 449.947,Z 512.534,A -85,B 0,C 180,E1 16305.239,E2 16305.239} C_VEL
LIN {X 0,Y 456.732,Z 521.124,A -85,B 0,C 180,E1 16302.424,E2 16302.424} C_VEL
LIN {X 0,Y 465.669,Z 533.115,A -85,B 0,C 180,E1 16299.107,E2 16299.107} C_VEL
LIN {X 0,Y 476.114,Z 547.561,A -85,B 0,C 180,E1 16295.695,E2 16295.695} C_VEL
LIN {X 0,Y 480.413,Z 553.943,A -85,B 0,C 180,E1 16294.4,E2 16294.4} C_VEL
LIN {X 0,Y 459.775,Z 769.066,A -85,B 0,C 180,E1 16290.718,E2 16290.718} C_VEL
LIN {X 0,Y 456.388,Z 799.137,A -85,B 0,C 180,E1 16290.123,E2 16290.123} C_VEL
LIN {X 0,Y 452.921,Z 822.388,A -85,B 0,C 180,E1 16289.521,E2 16289.521} C_VEL
LIN {X 0,Y 448.39,Z 847.377,A -85,B 0,C 180,E1 16288.714,E2 16288.714} C_VEL
LIN {X 0,Y 442.335,Z 874.588,A -85,B 0,C 180,E1 16287.622,E2 16287.622} C_VEL
LIN {X 0,Y 436.734,Z 896.25,A -85,B 0,C 180,E1 16286.577,E2 16286.577} C_VEL
LIN {X 0,Y 430.373,Z 918.242,A -85,B 0,C 180,E1 16285.336,E2 16285.336} C_VEL
LIN {X 0,Y 421.949,Z 944.101,A -85,B 0,C 180,E1 16283.606,E2 16283.606} C_VEL
LIN {X 0,Y 414.395,Z 964.899,A -85,B 0,C 180,E1 16281.955,E2 16281.955} C_VEL
LIN {X 0,Y 407.4,Z 982.782,A -85,B 0,C 180,E1 16280.329,E2 16280.329} C_VEL
LIN {X 0,Y 399.263,Z 1002.293,A -85,B 0,C 180,E1 16278.294,E2 16278.294} C_VEL
LIN {X 0,Y 389.935,Z 1022.959,A -85,B 0,C 180,E1 16275.749,E2 16275.749} C_VEL
LIN {X 0,Y 382.618,Z 1038.294,A -85,B 0,C 180,E1 16273.553,E2 16273.553} C_VEL
LIN {X 0,Y 375.796,Z 1052.098,A -85,B 0,C 180,E1 16271.302,E2 16271.302} C_VEL
